QRS_NEXT_CUT()
PTP {E1 29336.919,E2 29336.919}
PTP {X 0,Y 607.923,A -85,B 0,C 180,E1 29336.919,E2 29336.919,E3 0,E4 0,E5 0,E6 0}
QRS_SPEED_INIT()
LIN {X 0,Y 607.923,Z 862.5,A -85,B 0,C 180,E1 29336.919,E2 29336.919,E3 0,E4 0,E5 0,E6 0} C_VEL
LIN {X 0,Y 607.923,Z 712.094,A -85,B 0,C 180,E1 29336.919,E2 29336.919} C_VEL
LIN {X 0,Y 607.923,Z 704.209,A -85,B 0,C 180,E1 29336.919,E2 29336.919} C_VEL
LIN {X 0,Y 607.917,Z 702.213,A -85,B 0,C 180,E1 29336.718,E2 29336.718} C_VEL
LIN {X 0,Y 607.918,Z 702.326,A -85,B 0,C 180,E1 29335.353,E2 29335.353} C_VEL
LIN {X 0,Y 607.916,Z 700.521,A -85,B 0,C 180,E1 29333.863,E2 29333.863} C_VEL
LIN {X 0,Y 607.918,Z 696.809,A -85,B 0,C 180,E1 29332.439,E2 29332.439} C_VEL
LIN {X 0,Y 607.918,Z 691.472,A -85,B 0,C 180,E1 29331.106,E2 29331.106} C_VEL
LIN {X 0,Y 607.918,Z 684.642,A -85,B 0,C 180,E1 29329.864,E2 29329.864} C_VEL
LIN {X 0,Y 607.918,Z 676.351,A -85,B 0,C 180,E1 29328.713,E2 29328.713} C_VEL
LIN {X 0,Y 607.918,Z 666.686,A -85,B 0,C 180,E1 29327.654,E2 29327.654} C_VEL
LIN {X 0,Y 607.92,Z 654.876,A -85,B 0,C 180,E1 29326.639,E2 29326.639} C_VEL
LIN {X 0,Y 607.896,Z 641.663,A -85,B 0,C 180,E1 29325.765,E2 29325.765} C_VEL
LIN {X 0,Y 607.908,Z 627.971,A -85,B 0,C 180,E1 29325.084,E2 29325.084} C_VEL
LIN {X 0,Y 607.9,Z 613.71,A -85,B 0,C 180,E1 29324.571,E2 29324.571} C_VEL
LIN {X 0,Y 607.917,Z 598.614,A -85,B 0,C 180,E1 29324.222,E2 29324.222} C_VEL
LIN {X 0,Y 607.905,Z 485.578,A -85,B 0,C 180,E1 29322.865,E2 29322.865} C_VEL
LIN {X 0,Y 607.912,Z 437.987,A -85,B 0,C 180,E1 29319.693,E2 29319.693} C_VEL
LIN {X 0,Y 607.914,Z 390.758,A -85,B 0,C 180,E1 29316.493,E2 29316.493} C_VEL
LIN {X 0,Y 607.914,Z 343.309,A -85,B 0,C 180,E1 29313.214,E2 29313.214} C_VEL
LIN {X 0,Y 607.918,Z 297.198,A -85,B 0,C 180,E1 29309.949,E2 29309.949} C_VEL
LIN {X 0,Y 607.91,Z 256.209,A -85,B 0,C 180,E1 29307.015,E2 29307.015} C_VEL
LIN {X 0,Y 607.917,Z 237.015,A -85,B 0,C 180,E1 29305.685,E2 29305.685} C_VEL
LIN {X 0,Y 607.9,Z 237.013,A -85,B 0,C 180,E1 29302.514,E2 29302.514} C_VEL
LIN {X 0,Y 607.885,Z 237.014,A -85,B 0,C 180,E1 29299.167,E2 29299.167} C_VEL
LIN {X 0,Y 607.887,Z 237.015,A -85,B 0,C 180,E1 29296.09,E2 29296.09} C_VEL
LIN {X 0,Y 607.912,Z 237.016,A -85,B 0,C 180,E1 29292.916,E2 29292.916} C_VEL
LIN {X 0,Y 607.913,Z 237.011,A -85,B 0,C 180,E1 29289.655,E2 29289.655} C_VEL
LIN {X 0,Y 607.874,Z 237.015,A -85,B 0,C 180,E1 29286.454,E2 29286.454} C_VEL
LIN {X 0,Y 607.914,Z 237.101,A -85,B 0,C 180,E1 29285.87,E2 29285.87} C_VEL
LIN {X 0,Y 607.914,Z 274.11,A -85,B 0,C 180,E1 29282.76,E2 29282.76} C_VEL
LIN {X 0,Y 607.865,Z 300.482,A -85,B 0,C 180,E1 29280.62,E2 29280.62} C_VEL
LIN {X 0,Y 607.913,Z 528.733,A -85,B 0,C 180,E1 29277.674,E2 29277.674} C_VEL
LIN {X 0,Y 607.92,Z 562.49,A -85,B 0,C 180,E1 29277.209,E2 29277.209} C_VEL
LIN {X 0,Y 607.907,Z 582.621,A -85,B 0,C 180,E1 29276.76,E2 29276.76} C_VEL
LIN {X 0,Y 607.907,Z 601.981,A -85,B 0,C 180,E1 29276.155,E2 29276.155} C_VEL
LIN {X 0,Y 607.915,Z 621.48,A -85,B 0,C 180,E1 29275.37,E2 29275.37} C_VEL
LIN {X 0,Y 607.919,Z 640.204,A -85,B 0,C 180,E1 29274.434,E2 29274.434} C_VEL
LIN {X 0,Y 607.916,Z 658.169,A -85,B 0,C 180,E1 29273.352,E2 29273.352} C_VEL
LIN {X 0,Y 607.914,Z 675.868,A -85,B 0,C 180,E1 29272.075,E2 29272.075} C_VEL
LIN {X 0,Y 607.917,Z 692.721,A -85,B 0,C 180,E1 29270.633,E2 29270.633} C_VEL
LIN {X 0,Y 607.908,Z 707.84,A -85,B 0,C 180,E1 29269.106,E2 29269.106} C_VEL
LIN {X 0,Y 607.911,Z 721.188,A -85,B 0,C 180,E1 29267.517,E2 29267.517} C_VEL
LIN {X 0,Y 607.915,Z 733.113,A -85,B 0,C 180,E1 29265.845,E2 29265.845} C_VEL
LIN {X 0,Y 607.91,Z 743.612,A -85,B 0,C 180,E1 29264.089,E2 29264.089} C_VEL
LIN {X 0,Y 607.917,Z 752.375,A -85,B 0,C 180,E1 29262.318,E2 29262.318} C_VEL
LIN {X 0,Y 607.914,Z 759.869,A -85,B 0,C 180,E1 29260.424,E2 29260.424} C_VEL
LIN {X 0,Y 607.913,Z 765.53,A -85,B 0,C 180,E1 29258.513,E2 29258.513} C_VEL
LIN {X 0,Y 607.911,Z 769.46,A -85,B 0,C 180,E1 29256.611,E2 29256.611} C_VEL
LIN {X 0,Y 607.908,Z 771.826,A -85,B 0,C 180,E1 29254.623,E2 29254.623} C_VEL
LIN {X 0,Y 607.906,Z 772.455,A -85,B 0,C 180,E1 29252.734,E2 29252.734} C_VEL
LIN {X 0,Y 607.907,Z 771.512,A -85,B 0,C 180,E1 29250.848,E2 29250.848} C_VEL
LIN {X 0,Y 607.91,Z 768.741,A -85,B 0,C 180,E1 29248.869,E2 29248.869} C_VEL
LIN {X 0,Y 607.912,Z 764.424,A -85,B 0,C 180,E1 29246.983,E2 29246.983} C_VEL
LIN {X 0,Y 607.911,Z 758.417,A -85,B 0,C 180,E1 29245.094,E2 29245.094} C_VEL
LIN {X 0,Y 607.906,Z 751.044,A -85,B 0,C 180,E1 29243.294,E2 29243.294} C_VEL
LIN {X 0,Y 607.906,Z 741.815,A -85,B 0,C 180,E1 29241.487,E2 29241.487} C_VEL
LIN {X 0,Y 607.917,Z 731.146,A -85,B 0,C 180,E1 29239.768,E2 29239.768} C_VEL
LIN {X 0,Y 607.909,Z 719.138,A -85,B 0,C 180,E1 29238.135,E2 29238.135} C_VEL
LIN {X 0,Y 607.913,Z 704.904,A -85,B 0,C 180,E1 29236.494,E2 29236.494} C_VEL
LIN {X 0,Y 607.912,Z 688.936,A -85,B 0,C 180,E1 29234.938,E2 29234.938} C_VEL
LIN {X 0,Y 607.917,Z 672.324,A -85,B 0,C 180,E1 29233.567,E2 29233.567} C_VEL
LIN {X 0,Y 607.919,Z 654.646,A -85,B 0,C 180,E1 29232.335,E2 29232.335} C_VEL
LIN {X 0,Y 607.92,Z 636.895,A -85,B 0,C 180,E1 29231.293,E2 29231.293} C_VEL
LIN {X 0,Y 607.916,Z 617.178,A -85,B 0,C 180,E1 29230.345,E2 29230.345} C_VEL
LIN {X 0,Y 607.918,Z 598.54,A -85,B 0,C 180,E1 29229.636,E2 29229.636} C_VEL
LIN {X 0,Y 607.905,Z 579.176,A -85,B 0,C 180,E1 29229.064,E2 29229.064} C_VEL
LIN {X 0,Y 607.919,Z 559.341,A -85,B 0,C 180,E1 29228.648,E2 29228.648} C_VEL
LIN {X 0,Y 607.901,Z 304.548,A -85,B 0,C 180,E1 29225.345,E2 29225.345} C_VEL
LIN {X 0,Y 607.905,Z 299.084,A -85,B 0,C 180,E1 29225.262,E2 29225.262} C_VEL
LIN {X 0,Y 607.898,Z 255.446,A -85,B 0,C 180,E1 29222.196,E2 29222.196} C_VEL
LIN {X 0,Y 607.906,Z 237.013,A -85,B 0,C 180,E1 29220.853,E2 29220.853} C_VEL
LIN {X 0,Y 607.908,Z 237.015,A -85,B 0,C 180,E1 29217.575,E2 29217.575} C_VEL
LIN {X 0,Y 607.919,Z 237.015,A -85,B 0,C 180,E1 29214.16,E2 29214.16} C_VEL
LIN {X 0,Y 607.891,Z 237.015,A -85,B 0,C 180,E1 29210.953,E2 29210.953} C_VEL
LIN {X 0,Y 607.894,Z 237.015,A -85,B 0,C 180,E1 29207.85,E2 29207.85} C_VEL
LIN {X 0,Y 607.908,Z 237.015,A -85,B 0,C 180,E1 29204.721,E2 29204.721} C_VEL
LIN {X 0,Y 607.889,Z 237.015,A -85,B 0,C 180,E1 29201.519,E2 29201.519} C_VEL
LIN {X 0,Y 607.914,Z 237.013,A -85,B 0,C 180,E1 29198.442,E2 29198.442} C_VEL
LIN {X 0,Y 607.915,Z 237.015,A -85,B 0,C 180,E1 29195.146,E2 29195.146} C_VEL
LIN {X 0,Y 607.915,Z 237.012,A -85,B 0,C 180,E1 29191.868,E2 29191.868} C_VEL
LIN {X 0,Y 607.89,Z 237.015,A -85,B 0,C 180,E1 29188.704,E2 29188.704} C_VEL
LIN {X 0,Y 607.917,Z 237.094,A -85,B 0,C 180,E1 29185.735,E2 29185.735} C_VEL
LIN {X 0,Y 607.912,Z 269.505,A -85,B 0,C 180,E1 29183.25,E2 29183.25} C_VEL
LIN {X 0,Y 607.913,Z 310.074,A -85,B 0,C 180,E1 29180.106,E2 29180.106} C_VEL
LIN {X 0,Y 607.898,Z 351.534,A -85,B 0,C 180,E1 29176.975,E2 29176.975} C_VEL
LIN {X 0,Y 607.914,Z 393.877,A -85,B 0,C 180,E1 29173.846,E2 29173.846} C_VEL
LIN {X 0,Y 607.898,Z 436.137,A -85,B 0,C 180,E1 29170.788,E2 29170.788} C_VEL
LIN {X 0,Y 607.907,Z 578.351,A -85,B 0,C 180,E1 29169.061,E2 29169.061} C_VEL
LIN {X 0,Y 607.914,Z 594.993,A -85,B 0,C 180,E1 29168.677,E2 29168.677} C_VEL
LIN {X 0,Y 607.907,Z 610.686,A -85,B 0,C 180,E1 29168.132,E2 29168.132} C_VEL
LIN {X 0,Y 607.91,Z 625.671,A -85,B 0,C 180,E1 29167.419,E2 29167.419} C_VEL
LIN {X 0,Y 607.919,Z 639.478,A -85,B 0,C 180,E1 29166.576,E2 29166.576} C_VEL
LIN {X 0,Y 607.919,Z 652.518,A -85,B 0,C 180,E1 29165.569,E2 29165.569} C_VEL
LIN {X 0,Y 607.917,Z 664.366,A -85,B 0,C 180,E1 29164.434,E2 29164.434} C_VEL
LIN {X 0,Y 607.919,Z 674.596,A -85,B 0,C 180,E1 29163.206,E2 29163.206} C_VEL
LIN {X 0,Y 607.917,Z 683.39,A -85,B 0,C 180,E1 29161.885,E2 29161.885} C_VEL
LIN {X 0,Y 607.918,Z 690.67,A -85,B 0,C 180,E1 29160.472,E2 29160.472} C_VEL
LIN {X 0,Y 607.914,Z 696.343,A -85,B 0,C 180,E1 29158.964,E2 29158.964} C_VEL
LIN {X 0,Y 607.917,Z 700.143,A -85,B 0,C 180,E1 29157.455,E2 29157.455} C_VEL
LIN {X 0,Y 607.917,Z 702.102,A -85,B 0,C 180,E1 29155.945,E2 29155.945} C_VEL
LIN {X 0,Y 607.916,Z 702.384,A -85,B 0,C 180,E1 29154.432,E2 29154.432} C_VEL
LIN {X 0,Y 607.918,Z 700.91,A -85,B 0,C 180,E1 29152.915,E2 29152.915} C_VEL
LIN {X 0,Y 607.914,Z 697.651,A -85,B 0,C 180,E1 29151.392,E2 29151.392} C_VEL
LIN {X 0,Y 607.914,Z 692.883,A -85,B 0,C 180,E1 29149.96,E2 29149.96} C_VEL
LIN {X 0,Y 607.914,Z 686.165,A -85,B 0,C 180,E1 29148.521,E2 29148.521} C_VEL
LIN {X 0,Y 607.917,Z 677.957,A -85,B 0,C 180,E1 29147.172,E2 29147.172} C_VEL
LIN {X 0,Y 607.917,Z 668.253,A -85,B 0,C 180,E1 29145.912,E2 29145.912} C_VEL
LIN {X 0,Y 607.919,Z 656.49,A -85,B 0,C 180,E1 29144.694,E2 29144.694} C_VEL
LIN {X 0,Y 607.92,Z 644.082,A -85,B 0,C 180,E1 29143.666,E2 29143.666} C_VEL
LIN {X 0,Y 607.904,Z 629.927,A -85,B 0,C 180,E1 29142.73,E2 29142.73} C_VEL
LIN {X 0,Y 607.91,Z 615.562,A -85,B 0,C 180,E1 29141.989,E2 29141.989} C_VEL
LIN {X 0,Y 607.918,Z 600.152,A -85,B 0,C 180,E1 29141.393,E2 29141.393} C_VEL
LIN {X 0,Y 607.911,Z 584.62,A -85,B 0,C 180,E1 29140.97,E2 29140.97} C_VEL
LIN {X 0,Y 607.912,Z 567.42,A -85,B 0,C 180,E1 29140.696,E2 29140.696} C_VEL
LIN {X 0,Y 607.917,Z 435.757,A -85,B 0,C 180,E1 29139.101,E2 29139.101} C_VEL
LIN {X 0,Y 607.898,Z 392.014,A -85,B 0,C 180,E1 29135.927,E2 29135.927} C_VEL
LIN {X 0,Y 607.913,Z 348.895,A -85,B 0,C 180,E1 29132.738,E2 29132.738} C_VEL
LIN {X 0,Y 607.919,Z 306.939,A -85,B 0,C 180,E1 29129.564,E2 29129.564} C_VEL
LIN {X 0,Y 607.907,Z 266.15,A -85,B 0,C 180,E1 29126.396,E2 29126.396} C_VEL
LIN {X 0,Y 607.917,Z 246.516,A -85,B 0,C 180,E1 29124.912,E2 29124.912} C_VEL
LIN {X 0,Y 607.902,Z 237.015,A -85,B 0,C 180,E1 29124.252,E2 29124.252} C_VEL
LIN {X 0,Y 607.914,Z 237.013,A -85,B 0,C 180,E1 29121.075,E2 29121.075} C_VEL
LIN {X 0,Y 607.916,Z 237.209,A -85,B 0,C 180,E1 29119.151,E2 29119.151} C_VEL
LIN {X 0,Y 607.915,Z 286.021,A -85,B 0,C 180,E1 29116.132,E2 29116.132} C_VEL
LIN {X 0,Y 607.892,Z 298.558,A -85,B 0,C 180,E1 29115.28,E2 29115.28} C_VEL
LIN {X 0,Y 607.917,Z 306.589,A -85,B 0,C 180,E1 29114.534,E2 29114.534} C_VEL
LIN {X 0,Y 607.877,Z 311.103,A -85,B 0,C 180,E1 29113.91,E2 29113.91} C_VEL
LIN {X 0,Y 607.877,Z 312.629,A -85,B 0,C 180,E1 29113.436,E2 29113.436} C_VEL
LIN {X 0,Y 607.904,Z 312.223,A -85,B 0,C 180,E1 29113.091,E2 29113.091} C_VEL
LIN {X 0,Y 607.918,Z 310.278,A -85,B 0,C 180,E1 29112.787,E2 29112.787} C_VEL
LIN {X 0,Y 607.903,Z 306.612,A -85,B 0,C 180,E1 29112.532,E2 29112.532} C_VEL
LIN {X 0,Y 607.892,Z 300.365,A -85,B 0,C 180,E1 29112.337,E2 29112.337} C_VEL
LIN {X 0,Y 607.889,Z 290.203,A -85,B 0,C 180,E1 29112.246,E2 29112.246} C_VEL
LIN {X 0,Y 607.888,Z 237.014,A -85,B 0,C 180,E1 29112.229,E2 29112.229} C_VEL
LIN {X 0,Y 607.874,Z 237.015,A -85,B 0,C 180,E1 29109.221,E2 29109.221} C_VEL
LIN {X 0,Y 607.904,Z 237.171,A -85,B 0,C 180,E1 29106.191,E2 29106.191} C_VEL
LIN {X 0,Y 607.917,Z 288.408,A -85,B 0,C 180,E1 29103.158,E2 29103.158} C_VEL
LIN {X 0,Y 607.913,Z 302.276,A -85,B 0,C 180,E1 29102.369,E2 29102.369} C_VEL
LIN {X 0,Y 607.904,Z 524.18,A -85,B 0,C 180,E1 29099.377,E2 29099.377} C_VEL
LIN {X 0,Y 607.903,Z 608.537,A -85,B 0,C 180,E1 29098.234,E2 29098.234} C_VEL
LIN {X 0,Y 607.909,Z 629.043,A -85,B 0,C 180,E1 29097.785,E2 29097.785} C_VEL
LIN {X 0,Y 607.906,Z 649.64,A -85,B 0,C 180,E1 29097.18,E2 29097.18} C_VEL
LIN {X 0,Y 607.913,Z 669.578,A -85,B 0,C 180,E1 29096.417,E2 29096.417} C_VEL
LIN {X 0,Y 607.918,Z 690.744,A -85,B 0,C 180,E1 29095.422,E2 29095.422} C_VEL
LIN {X 0,Y 607.916,Z 710.11,A -85,B 0,C 180,E1 29094.331,E2 29094.331} C_VEL
LIN {X 0,Y 607.914,Z 728.559,A -85,B 0,C 180,E1 29093.096,E2 29093.096} C_VEL
LIN {X 0,Y 607.911,Z 746.777,A -85,B 0,C 180,E1 29091.678,E2 29091.678} C_VEL
LIN {X 0,Y 607.913,Z 763.653,A -85,B 0,C 180,E1 29090.156,E2 29090.156} C_VEL
LIN {X 0,Y 607.918,Z 779.465,A -85,B 0,C 180,E1 29088.508,E2 29088.508} C_VEL
LIN {X 0,Y 607.913,Z 793.413,A -85,B 0,C 180,E1 29086.817,E2 29086.817} C_VEL
LIN {X 0,Y 607.918,Z 805.901,A -85,B 0,C 180,E1 29085.062,E2 29085.062} C_VEL
LIN {X 0,Y 607.919,Z 817.421,A -85,B 0,C 180,E1 29083.176,E2 29083.176} C_VEL
LIN {X 0,Y 607.912,Z 827.061,A -85,B 0,C 180,E1 29081.287,E2 29081.287} C_VEL
LIN {X 0,Y 607.911,Z 835.464,A -85,B 0,C 180,E1 29079.276,E2 29079.276} C_VEL
LIN {X 0,Y 607.91,Z 842.129,A -85,B 0,C 180,E1 29077.276,E2 29077.276} C_VEL
LIN {X 0,Y 607.912,Z 847.015,A -85,B 0,C 180,E1 29075.285,E2 29075.285} C_VEL
LIN {X 0,Y 607.917,Z 850.447,A -85,B 0,C 180,E1 29073.206,E2 29073.206} C_VEL
LIN {X 0,Y 607.91,Z 852.21,A -85,B 0,C 180,E1 29071.225,E2 29071.225} C_VEL
LIN {X 0,Y 607.902,Z 852.329,A -85,B 0,C 180,E1 29069.246,E2 29069.246} C_VEL
LIN {X 0,Y 607.908,Z 850.896,A -85,B 0,C 180,E1 29067.172,E2 29067.172} C_VEL
LIN {X 0,Y 607.912,Z 847.987,A -85,B 0,C 180,E1 29065.188,E2 29065.188} C_VEL
LIN {X 0,Y 607.915,Z 843.399,A -85,B 0,C 180,E1 29063.199,E2 29063.199} C_VEL
LIN {X 0,Y 607.906,Z 837.238,A -85,B 0,C 180,E1 29061.201,E2 29061.201} C_VEL
LIN {X 0,Y 607.899,Z 829.657,A -85,B 0,C 180,E1 29059.289,E2 29059.289} C_VEL
LIN {X 0,Y 607.899,Z 820.326,A -85,B 0,C 180,E1 29057.364,E2 29057.364} C_VEL
LIN {X 0,Y 607.904,Z 809.744,A -85,B 0,C 180,E1 29055.522,E2 29055.522} C_VEL
LIN {X 0,Y 607.913,Z 797.033,A -85,B 0,C 180,E1 29053.665,E2 29053.665} C_VEL
LIN {X 0,Y 607.907,Z 782.865,A -85,B 0,C 180,E1 29051.889,E2 29051.889} C_VEL
LIN {X 0,Y 607.91,Z 767.096,A -85,B 0,C 180,E1 29050.185,E2 29050.185} C_VEL
LIN {X 0,Y 607.918,Z 750.497,A -85,B 0,C 180,E1 29048.635,E2 29048.635} C_VEL
LIN {X 0,Y 607.913,Z 732.133,A -85,B 0,C 180,E1 29047.16,E2 29047.16} C_VEL
LIN {X 0,Y 607.915,Z 713.681,A -85,B 0,C 180,E1 29045.898,E2 29045.898} C_VEL
LIN {X 0,Y 607.918,Z 693.554,A -85,B 0,C 180,E1 29044.726,E2 29044.726} C_VEL
LIN {X 0,Y 607.904,Z 674.553,A -85,B 0,C 180,E1 29043.792,E2 29043.792} C_VEL
LIN {X 0,Y 607.906,Z 653.962,A -85,B 0,C 180,E1 29042.976,E2 29042.976} C_VEL
LIN {X 0,Y 607.917,Z 632.86,A -85,B 0,C 180,E1 29042.313,E2 29042.313} C_VEL
LIN {X 0,Y 607.905,Z 613.424,A -85,B 0,C 180,E1 29041.861,E2 29041.861} C_VEL
LIN {X 0,Y 607.918,Z 585.551,A -85,B 0,C 180,E1 29041.436,E2 29041.436} C_VEL
LIN {X 0,Y 607.876,Z 362.254,A -85,B 0,C 180,E1 29038.447,E2 29038.447} C_VEL
LIN {X 0,Y 607.915,Z 302.732,A -85,B 0,C 180,E1 29037.631,E2 29037.631} C_VEL
LIN {X 0,Y 607.898,Z 258.862,A -85,B 0,C 180,E1 29034.622,E2 29034.622} C_VEL
LIN {X 0,Y 607.893,Z 237.014,A -85,B 0,C 180,E1 29033.07,E2 29033.07} C_VEL
LIN {X 0,Y 607.882,Z 237.015,A -85,B 0,C 180,E1 29029.974,E2 29029.974} C_VEL
LIN {X 0,Y 607.902,Z 237.013,A -85,B 0,C 180,E1 29027.753,E2 29027.753} C_VEL
LIN {X 0,Y 607.902,Z 333.704,A -85,B 0,C 180,E1 29027.733,E2 29027.733} C_VEL
LIN {X 0,Y 607.904,Z 341.134,A -85,B 0,C 180,E1 29027.596,E2 29027.596} C_VEL
LIN {X 0,Y 607.909,Z 345.398,A -85,B 0,C 180,E1 29027.402,E2 29027.402} C_VEL
LIN {X 0,Y 607.917,Z 347.912,A -85,B 0,C 180,E1 29027.184,E2 29027.184} C_VEL
LIN {X 0,Y 607.917,Z 349.732,A -85,B 0,C 180,E1 29026.826,E2 29026.826} C_VEL
LIN {X 0,Y 607.884,Z 349.905,A -85,B 0,C 180,E1 29026.434,E2 29026.434} C_VEL
LIN {X 0,Y 607.884,Z 348.098,A -85,B 0,C 180,E1 29025.912,E2 29025.912} C_VEL
LIN {X 0,Y 607.915,Z 343.085,A -85,B 0,C 180,E1 29025.199,E2 29025.199} C_VEL
LIN {X 0,Y 607.899,Z 335.413,A -85,B 0,C 180,E1 29024.452,E2 29024.452} C_VEL
LIN {X 0,Y 607.906,Z 321.424,A -85,B 0,C 180,E1 29023.433,E2 29023.433} C_VEL
LIN {X 0,Y 607.911,Z 279.23,A -85,B 0,C 180,E1 29020.459,E2 29020.459} C_VEL
LIN {X 0,Y 607.895,Z 240.537,A -85,B 0,C 180,E1 29017.605,E2 29017.605} C_VEL
LIN {X 0,Y 607.917,Z 237.015,A -85,B 0,C 180,E1 29017.336,E2 29017.336} C_VEL
LIN {X 0,Y 607.89,Z 237.014,A -85,B 0,C 180,E1 29014.173,E2 29014.173} C_VEL
LIN {X 0,Y 607.911,Z 237.007,A -85,B 0,C 180,E1 29010.874,E2 29010.874} C_VEL
LIN {X 0,Y 607.873,Z 237.012,A -85,B 0,C 180,E1 29007.742,E2 29007.742} C_VEL
LIN {X 0,Y 607.866,Z 237.166,A -85,B 0,C 180,E1 29006.08,E2 29006.08} C_VEL
LIN {X 0,Y 607.91,Z 268.682,A -85,B 0,C 180,E1 29004.021,E2 29004.021} C_VEL
LIN {X 0,Y 607.911,Z 313.328,A -85,B 0,C 180,E1 29000.809,E2 29000.809} C_VEL
LIN {X 0,Y 607.913,Z 359.543,A -85,B 0,C 180,E1 28997.566,E2 28997.566} C_VEL
LIN {X 0,Y 607.912,Z 407.398,A -85,B 0,C 180,E1 28994.283,E2 28994.283} C_VEL
LIN {X 0,Y 607.915,Z 454.742,A -85,B 0,C 180,E1 28991.095,E2 28991.095} C_VEL
LIN {X 0,Y 607.91,Z 485.669,A -85,B 0,C 180,E1 28989.043,E2 28989.043} C_VEL
LIN {X 0,Y 607.919,Z 599.073,A -85,B 0,C 180,E1 28987.679,E2 28987.679} C_VEL
LIN {X 0,Y 607.903,Z 613.667,A -85,B 0,C 180,E1 28987.34,E2 28987.34} C_VEL
LIN {X 0,Y 607.908,Z 627.464,A -85,B 0,C 180,E1 28986.848,E2 28986.848} C_VEL
LIN {X 0,Y 607.897,Z 640.982,A -85,B 0,C 180,E1 28986.184,E2 28986.184} C_VEL
LIN {X 0,Y 607.918,Z 654.051,A -85,B 0,C 180,E1 28985.332,E2 28985.332} C_VEL
LIN {X 0,Y 607.919,Z 665.313,A -85,B 0,C 180,E1 28984.386,E2 28984.386} C_VEL
LIN {X 0,Y 607.917,Z 674.746,A -85,B 0,C 180,E1 28983.394,E2 28983.394} C_VEL
LIN {X 0,Y 607.918,Z 683.863,A -85,B 0,C 180,E1 28982.168,E2 28982.168} C_VEL
LIN {X 0,Y 607.918,Z 690.803,A -85,B 0,C 180,E1 28980.942,E2 28980.942} C_VEL
LIN {X 0,Y 607.919,Z 696.321,A -85,B 0,C 180,E1 28979.623,E2 28979.623} C_VEL
LIN {X 0,Y 607.916,Z 700.179,A -85,B 0,C 180,E1 28978.209,E2 28978.209} C_VEL
LIN {X 0,Y 607.916,Z 702.093,A -85,B 0,C 180,E1 28976.888,E2 28976.888} C_VEL
LIN {X 0,Y 607.917,Z 702.213,A -85,B 0,C 180,E1 28976.718,E2 28976.718} C_VEL
LIN {X 0,Y 606.916,Z 702.497,A -85,B 0,C 180,E1 28975.992,E2 28975.992} C_VEL
LIN {X 0,Y 602.995,Z 701.936,A -85,B 0,C 180,E1 28974.831,E2 28974.831} C_VEL
LIN {X 0,Y 600.268,Z 700.564,A -85,B 0,C 180,E1 28973.859,E2 28973.859} C_VEL
LIN {X 0,Y 599.917,Z 699.685,A -85,B 0,C 180,E1 28973.441,E2 28973.441} C_VEL
LIN {X 0,Y 599.916,Z 695.635,A -85,B 0,C 180,E1 28972.048,E2 28972.048} C_VEL
LIN {X 0,Y 599.922,Z 689.797,A -85,B 0,C 180,E1 28970.696,E2 28970.696} C_VEL
LIN {X 0,Y 599.932,Z 682.383,A -85,B 0,C 180,E1 28969.436,E2 28969.436} C_VEL
LIN {X 0,Y 599.948,Z 673.454,A -85,B 0,C 180,E1 28968.268,E2 28968.268} C_VEL
LIN {X 0,Y 599.971,Z 663.013,A -85,B 0,C 180,E1 28967.194,E2 28967.194} C_VEL
LIN {X 0,Y 599.986,Z 650.76,A -85,B 0,C 180,E1 28966.213,E2 28966.213} C_VEL
LIN {X 0,Y 600.002,Z 638.006,A -85,B 0,C 180,E1 28965.426,E2 28965.426} C_VEL
LIN {X 0,Y 600.029,Z 624.106,A -85,B 0,C 180,E1 28964.779,E2 28964.779} C_VEL
LIN {X 0,Y 600.056,Z 609.272,A -85,B 0,C 180,E1 28964.296,E2 28964.296} C_VEL
LIN {X 0,Y 600.085,Z 594.128,A -85,B 0,C 180,E1 28963.999,E2 28963.999} C_VEL
LIN {X 0,Y 600.045,Z 485.282,A -85,B 0,C 180,E1 28962.671,E2 28962.671} C_VEL
LIN {X 0,Y 600.129,Z 438.627,A -85,B 0,C 180,E1 28959.52,E2 28959.52} C_VEL
LIN {X 0,Y 600.229,Z 391.488,A -85,B 0,C 180,E1 28956.285,E2 28956.285} C_VEL
LIN {X 0,Y 600.333,Z 343.943,A -85,B 0,C 180,E1 28952.955,E2 28952.955} C_VEL
LIN {X 0,Y 600.463,Z 298.529,A -85,B 0,C 180,E1 28949.699,E2 28949.699} C_VEL
LIN {X 0,Y 600.322,Z 250.637,A -85,B 0,C 180,E1 28946.315,E2 28946.315} C_VEL
LIN {X 0,Y 600.245,Z 239.331,A -85,B 0,C 180,E1 28945.543,E2 28945.543} C_VEL
LIN {X 0,Y 599.953,Z 238.005,A -85,B 0,C 180,E1 28945.415,E2 28945.415} C_VEL
LIN {X 0,Y 599.96,Z 238,A -85,B 0,C 180,E1 28942.293,E2 28942.293} C_VEL
LIN {X 0,Y 599.952,Z 238.003,A -85,B 0,C 180,E1 28938.956,E2 28938.956} C_VEL
LIN {X 0,Y 599.976,Z 238.004,A -85,B 0,C 180,E1 28935.775,E2 28935.775} C_VEL
LIN {X 0,Y 599.951,Z 238.004,A -85,B 0,C 180,E1 28932.555,E2 28932.555} C_VEL
LIN {X 0,Y 599.959,Z 238.002,A -85,B 0,C 180,E1 28929.17,E2 28929.17} C_VEL
LIN {X 0,Y 599.959,Z 238.135,A -85,B 0,C 180,E1 28926.273,E2 28926.273} C_VEL
LIN {X 0,Y 600.701,Z 241.601,A -85,B 0,C 180,E1 28925.926,E2 28925.926} C_VEL
LIN {X 0,Y 600.543,Z 278.735,A -85,B 0,C 180,E1 28922.776,E2 28922.776} C_VEL
LIN {X 0,Y 600.532,Z 300.692,A -85,B 0,C 180,E1 28920.985,E2 28920.985} C_VEL
LIN {X 0,Y 600.761,Z 314.388,A -85,B 0,C 180,E1 28920.792,E2 28920.792} C_VEL
LIN {X 0,Y 600.62,Z 561.056,A -85,B 0,C 180,E1 28917.551,E2 28917.551} C_VEL
LIN {X 0,Y 600.559,Z 581.248,A -85,B 0,C 180,E1 28917.104,E2 28917.104} C_VEL
LIN {X 0,Y 600.497,Z 601.492,A -85,B 0,C 180,E1 28916.476,E2 28916.476} C_VEL
LIN {X 0,Y 600.424,Z 621.676,A -85,B 0,C 180,E1 28915.656,E2 28915.656} C_VEL
LIN {X 0,Y 600.344,Z 640.35,A -85,B 0,C 180,E1 28914.711,E2 28914.711} C_VEL
LIN {X 0,Y 600.274,Z 658.008,A -85,B 0,C 180,E1 28913.634,E2 28913.634} C_VEL
LIN {X 0,Y 600.199,Z 675.975,A -85,B 0,C 180,E1 28912.323,E2 28912.323} C_VEL
LIN {X 0,Y 600.123,Z 692.516,A -85,B 0,C 180,E1 28910.888,E2 28910.888} C_VEL
LIN {X 0,Y 600.061,Z 707.447,A -85,B 0,C 180,E1 28909.365,E2 28909.365} C_VEL
LIN {X 0,Y 600.006,Z 720.857,A -85,B 0,C 180,E1 28907.756,E2 28907.756} C_VEL
LIN {X 0,Y 599.976,Z 732.845,A -85,B 0,C 180,E1 28906.06,E2 28906.06} C_VEL
LIN {X 0,Y 599.948,Z 743.391,A -85,B 0,C 180,E1 28904.28,E2 28904.28} C_VEL
LIN {X 0,Y 599.929,Z 752.089,A -85,B 0,C 180,E1 28902.513,E2 28902.513} C_VEL
LIN {X 0,Y 599.923,Z 759.729,A -85,B 0,C 180,E1 28900.564,E2 28900.564} C_VEL
LIN {X 0,Y 599.917,Z 765.422,A -85,B 0,C 180,E1 28898.627,E2 28898.627} C_VEL
LIN {X 0,Y 599.914,Z 769.398,A -85,B 0,C 180,E1 28896.7,E2 28896.7} C_VEL
LIN {X 0,Y 599.91,Z 771.811,A -85,B 0,C 180,E1 28894.668,E2 28894.668} C_VEL
LIN {X 0,Y 599.907,Z 772.466,A -85,B 0,C 180,E1 28892.77,E2 28892.77} C_VEL
LIN {X 0,Y 599.904,Z 771.452,A -85,B 0,C 180,E1 28890.764,E2 28890.764} C_VEL
LIN {X 0,Y 599.91,Z 768.805,A -85,B 0,C 180,E1 28888.854,E2 28888.854} C_VEL
LIN {X 0,Y 599.914,Z 764.532,A -85,B 0,C 180,E1 28886.943,E2 28886.943} C_VEL
LIN {X 0,Y 599.921,Z 758.565,A -85,B 0,C 180,E1 28885.028,E2 28885.028} C_VEL
LIN {X 0,Y 599.925,Z 751.236,A -85,B 0,C 180,E1 28883.204,E2 28883.204} C_VEL
LIN {X 0,Y 599.94,Z 742.034,A -85,B 0,C 180,E1 28881.373,E2 28881.373} C_VEL
LIN {X 0,Y 599.977,Z 731.414,A -85,B 0,C 180,E1 28879.631,E2 28879.631} C_VEL
LIN {X 0,Y 600.011,Z 719.467,A -85,B 0,C 180,E1 28877.977,E2 28877.977} C_VEL
LIN {X 0,Y 600.067,Z 705.293,A -85,B 0,C 180,E1 28876.314,E2 28876.314} C_VEL
LIN {X 0,Y 600.128,Z 689.941,A -85,B 0,C 180,E1 28874.787,E2 28874.787} C_VEL
LIN {X 0,Y 600.205,Z 673.528,A -85,B 0,C 180,E1 28873.399,E2 28873.399} C_VEL
LIN {X 0,Y 600.288,Z 656.096,A -85,B 0,C 180,E1 28872.153,E2 28872.153} C_VEL
LIN {X 0,Y 600.367,Z 637.68,A -85,B 0,C 180,E1 28871.049,E2 28871.049} C_VEL
LIN {X 0,Y 600.439,Z 618.129,A -85,B 0,C 180,E1 28870.09,E2 28870.09} C_VEL
LIN {X 0,Y 600.509,Z 599.057,A -85,B 0,C 180,E1 28869.349,E2 28869.349} C_VEL
LIN {X 0,Y 600.563,Z 578.722,A -85,B 0,C 180,E1 28868.741,E2 28868.741} C_VEL
LIN {X 0,Y 600.621,Z 558.236,A -85,B 0,C 180,E1 28868.316,E2 28868.316} C_VEL
LIN {X 0,Y 600.809,Z 305.225,A -85,B 0,C 180,E1 28864.999,E2 28864.999} C_VEL
LIN {X 0,Y 600.554,Z 299.244,A -85,B 0,C 180,E1 28864.905,E2 28864.905} C_VEL
LIN {X 0,Y 600.676,Z 255.491,A -85,B 0,C 180,E1 28861.788,E2 28861.788} C_VEL
LIN {X 0,Y 600.531,Z 240.103,A -85,B 0,C 180,E1 28860.656,E2 28860.656} C_VEL
LIN {X 0,Y 599.979,Z 238.001,A -85,B 0,C 180,E1 28860.443,E2 28860.443} C_VEL
LIN {X 0,Y 599.953,Z 238.004,A -85,B 0,C 180,E1 28857.312,E2 28857.312} C_VEL
LIN {X 0,Y 599.975,Z 238.005,A -85,B 0,C 180,E1 28854.083,E2 28854.083} C_VEL
LIN {X 0,Y 599.952,Z 238.005,A -85,B 0,C 180,E1 28850.952,E2 28850.952} C_VEL
LIN {X 0,Y 599.953,Z 238.004,A -85,B 0,C 180,E1 28847.807,E2 28847.807} C_VEL
LIN {X 0,Y 599.976,Z 238.004,A -85,B 0,C 180,E1 28844.635,E2 28844.635} C_VEL
LIN {X 0,Y 599.961,Z 238.003,A -85,B 0,C 180,E1 28841.27,E2 28841.27} C_VEL
LIN {X 0,Y 599.978,Z 238,A -85,B 0,C 180,E1 28838.069,E2 28838.069} C_VEL
LIN {X 0,Y 599.965,Z 238.003,A -85,B 0,C 180,E1 28834.864,E2 28834.864} C_VEL
LIN {X 0,Y 599.973,Z 238.004,A -85,B 0,C 180,E1 28831.553,E2 28831.553} C_VEL
LIN {X 0,Y 599.953,Z 238.004,A -85,B 0,C 180,E1 28828.358,E2 28828.358} C_VEL
LIN {X 0,Y 599.981,Z 238.047,A -85,B 0,C 180,E1 28825.995,E2 28825.995} C_VEL
LIN {X 0,Y 600.345,Z 242.342,A -85,B 0,C 180,E1 28825.66,E2 28825.66} C_VEL
LIN {X 0,Y 600.484,Z 284.835,A -85,B 0,C 180,E1 28822.415,E2 28822.415} C_VEL
LIN {X 0,Y 600.35,Z 325.484,A -85,B 0,C 180,E1 28819.255,E2 28819.255} C_VEL
LIN {X 0,Y 600.255,Z 367.017,A -85,B 0,C 180,E1 28816.102,E2 28816.102} C_VEL
LIN {X 0,Y 600.148,Z 409.648,A -85,B 0,C 180,E1 28812.934,E2 28812.934} C_VEL
LIN {X 0,Y 600.155,Z 436.538,A -85,B 0,C 180,E1 28810.993,E2 28810.993} C_VEL
LIN {X 0,Y 600.143,Z 578.774,A -85,B 0,C 180,E1 28809.24,E2 28809.24} C_VEL
LIN {X 0,Y 600.129,Z 595.596,A -85,B 0,C 180,E1 28808.842,E2 28808.842} C_VEL
LIN {X 0,Y 600.088,Z 611.149,A -85,B 0,C 180,E1 28808.287,E2 28808.287} C_VEL
LIN {X 0,Y 600.053,Z 627.239,A -85,B 0,C 180,E1 28807.499,E2 28807.499} C_VEL
LIN {X 0,Y 600.024,Z 641.272,A -85,B 0,C 180,E1 28806.603,E2 28806.603} C_VEL
LIN {X 0,Y 599.992,Z 655.087,A -85,B 0,C 180,E1 28805.485,E2 28805.485} C_VEL
LIN {X 0,Y 599.962,Z 666.654,A -85,B 0,C 180,E1 28804.301,E2 28804.301} C_VEL
LIN {X 0,Y 599.942,Z 676.488,A -85,B 0,C 180,E1 28803.057,E2 28803.057} C_VEL
LIN {X 0,Y 599.927,Z 684.842,A -85,B 0,C 180,E1 28801.719,E2 28801.719} C_VEL
LIN {X 0,Y 599.92,Z 691.759,A -85,B 0,C 180,E1 28800.287,E2 28800.287} C_VEL
LIN {X 0,Y 599.916,Z 697.135,A -85,B 0,C 180,E1 28798.759,E2 28798.759} C_VEL
LIN {X 0,Y 599.915,Z 700.568,A -85,B 0,C 180,E1 28797.23,E2 28797.23} C_VEL
LIN {X 0,Y 599.914,Z 702.345,A -85,B 0,C 180,E1 28795.603,E2 28795.603} C_VEL
LIN {X 0,Y 599.915,Z 702.177,A -85,B 0,C 180,E1 28794.069,E2 28794.069} C_VEL
LIN {X 0,Y 599.915,Z 700.322,A -85,B 0,C 180,E1 28792.531,E2 28792.531} C_VEL
LIN {X 0,Y 599.916,Z 696.636,A -85,B 0,C 180,E1 28790.987,E2 28790.987} C_VEL
LIN {X 0,Y 599.919,Z 691.338,A -85,B 0,C 180,E1 28789.525,E2 28789.525} C_VEL
LIN {X 0,Y 599.929,Z 684.221,A -85,B 0,C 180,E1 28788.074,E2 28788.074} C_VEL
LIN {X 0,Y 599.945,Z 675.393,A -85,B 0,C 180,E1 28786.704,E2 28786.704} C_VEL
LIN {X 0,Y 599.965,Z 665.048,A -85,B 0,C 180,E1 28785.425,E2 28785.425} C_VEL
LIN {X 0,Y 599.995,Z 652.968,A -85,B 0,C 180,E1 28784.239,E2 28784.239} C_VEL
LIN {X 0,Y 600.024,Z 640.4,A -85,B 0,C 180,E1 28783.245,E2 28783.245} C_VEL
LIN {X 0,Y 600.054,Z 626.791,A -85,B 0,C 180,E1 28782.387,E2 28782.387} C_VEL
LIN {X 0,Y 600.086,Z 611.637,A -85,B 0,C 180,E1 28781.645,E2 28781.645} C_VEL
LIN {X 0,Y 600.129,Z 596.071,A -85,B 0,C 180,E1 28781.083,E2 28781.083} C_VEL
LIN {X 0,Y 600.145,Z 579.592,A -85,B 0,C 180,E1 28780.685,E2 28780.685} C_VEL
LIN {X 0,Y 600.176,Z 538.532,A -85,B 0,C 180,E1 28780.158,E2 28780.158} C_VEL
LIN {X 0,Y 600.114,Z 436,A -85,B 0,C 180,E1 28778.907,E2 28778.907} C_VEL
LIN {X 0,Y 600.182,Z 393.117,A -85,B 0,C 180,E1 28775.755,E2 28775.755} C_VEL
LIN {X 0,Y 600.295,Z 350.929,A -85,B 0,C 180,E1 28772.595,E2 28772.595} C_VEL
LIN {X 0,Y 600.415,Z 308.75,A -85,B 0,C 180,E1 28769.365,E2 28769.365} C_VEL
LIN {X 0,Y 600.429,Z 271.807,A -85,B 0,C 180,E1 28766.494,E2 28766.494} C_VEL
LIN {X 0,Y 599.96,Z 238.004,A -85,B 0,C 180,E1 28764.171,E2 28764.171} C_VEL
LIN {X 0,Y 599.978,Z 238.001,A -85,B 0,C 180,E1 28760.95,E2 28760.95} C_VEL
LIN {X 0,Y 599.977,Z 238.162,A -85,B 0,C 180,E1 28759.738,E2 28759.738} C_VEL
LIN {X 0,Y 601.386,Z 241.742,A -85,B 0,C 180,E1 28759.391,E2 28759.391} C_VEL
LIN {X 0,Y 601.191,Z 290.6,A -85,B 0,C 180,E1 28756.341,E2 28756.341} C_VEL
LIN {X 0,Y 601.878,Z 304.835,A -85,B 0,C 180,E1 28755.423,E2 28755.423} C_VEL
LIN {X 0,Y 602.923,Z 312.502,A -85,B 0,C 180,E1 28754.784,E2 28754.784} C_VEL
LIN {X 0,Y 603.87,Z 317.346,A -85,B 0,C 180,E1 28754.193,E2 28754.193} C_VEL
LIN {X 0,Y 604.594,Z 319.521,A -85,B 0,C 180,E1 28753.723,E2 28753.723} C_VEL
LIN {X 0,Y 605.181,Z 320.146,A -85,B 0,C 180,E1 28753.231,E2 28753.231} C_VEL
LIN {X 0,Y 605.41,Z 318.965,A -85,B 0,C 180,E1 28752.749,E2 28752.749} C_VEL
LIN {X 0,Y 605.162,Z 316.09,A -85,B 0,C 180,E1 28752.337,E2 28752.337} C_VEL
LIN {X 0,Y 604.488,Z 311.563,A -85,B 0,C 180,E1 28752.011,E2 28752.011} C_VEL
LIN {X 0,Y 603.535,Z 305.051,A -85,B 0,C 180,E1 28751.795,E2 28751.795} C_VEL
LIN {X 0,Y 602.626,Z 294.653,A -85,B 0,C 180,E1 28751.692,E2 28751.692} C_VEL
LIN {X 0,Y 602.377,Z 242.797,A -85,B 0,C 180,E1 28751.665,E2 28751.665} C_VEL
LIN {X 0,Y 600.469,Z 239.953,A -85,B 0,C 180,E1 28751.46,E2 28751.46} C_VEL
LIN {X 0,Y 599.973,Z 238.003,A -85,B 0,C 180,E1 28751.389,E2 28751.389} C_VEL
LIN {X 0,Y 599.94,Z 238.005,A -85,B 0,C 180,E1 28748.193,E2 28748.193} C_VEL
LIN {X 0,Y 599.98,Z 238.019,A -85,B 0,C 180,E1 28746.694,E2 28746.694} C_VEL
LIN {X 0,Y 601.097,Z 241.818,A -85,B 0,C 180,E1 28746.382,E2 28746.382} C_VEL
LIN {X 0,Y 600.926,Z 292.429,A -85,B 0,C 180,E1 28743.358,E2 28743.358} C_VEL
LIN {X 0,Y 601.014,Z 302.701,A -85,B 0,C 180,E1 28742.781,E2 28742.781} C_VEL
LIN {X 0,Y 600.96,Z 495.848,A -85,B 0,C 180,E1 28740.133,E2 28740.133} C_VEL
LIN {X 0,Y 600.847,Z 608.558,A -85,B 0,C 180,E1 28738.596,E2 28738.596} C_VEL
LIN {X 0,Y 600.79,Z 629.726,A -85,B 0,C 180,E1 28738.126,E2 28738.126} C_VEL
LIN {X 0,Y 600.703,Z 651.089,A -85,B 0,C 180,E1 28737.481,E2 28737.481} C_VEL
LIN {X 0,Y 600.638,Z 671.563,A -85,B 0,C 180,E1 28736.68,E2 28736.68} C_VEL
LIN {X 0,Y 600.538,Z 691.744,A -85,B 0,C 180,E1 28735.704,E2 28735.704} C_VEL
LIN {X 0,Y 600.434,Z 710.925,A -85,B 0,C 180,E1 28734.602,E2 28734.602} C_VEL
LIN {X 0,Y 600.348,Z 730.016,A -85,B 0,C 180,E1 28733.3,E2 28733.3} C_VEL
LIN {X 0,Y 600.246,Z 747.555,A -85,B 0,C 180,E1 28731.903,E2 28731.903} C_VEL
LIN {X 0,Y 600.16,Z 765.176,A -85,B 0,C 180,E1 28730.275,E2 28730.275} C_VEL
LIN {X 0,Y 600.091,Z 780.318,A -85,B 0,C 180,E1 28728.657,E2 28728.657} C_VEL
LIN {X 0,Y 600.038,Z 794.885,A -85,B 0,C 180,E1 28726.855,E2 28726.855} C_VEL
LIN {X 0,Y 599.994,Z 807.187,A -85,B 0,C 180,E1 28725.068,E2 28725.068} C_VEL
LIN {X 0,Y 599.956,Z 818.772,A -85,B 0,C 180,E1 28723.1,E2 28723.1} C_VEL
LIN {X 0,Y 599.94,Z 828.43,A -85,B 0,C 180,E1 28721.147,E2 28721.147} C_VEL
LIN {X 0,Y 599.928,Z 836.176,A -85,B 0,C 180,E1 28719.207,E2 28719.207} C_VEL
LIN {X 0,Y 599.922,Z 842.894,A -85,B 0,C 180,E1 28717.084,E2 28717.084} C_VEL
LIN {X 0,Y 599.917,Z 847.635,A -85,B 0,C 180,E1 28715.068,E2 28715.068} C_VEL
LIN {X 0,Y 599.914,Z 850.786,A -85,B 0,C 180,E1 28712.962,E2 28712.962} C_VEL
LIN {X 0,Y 599.903,Z 852.332,A -85,B 0,C 180,E1 28710.764,E2 28710.764} C_VEL
LIN {X 0,Y 599.907,Z 852.209,A -85,B 0,C 180,E1 28708.758,E2 28708.758} C_VEL
LIN {X 0,Y 599.916,Z 850.373,A -85,B 0,C 180,E1 28706.686,E2 28706.686} C_VEL
LIN {X 0,Y 599.915,Z 846.812,A -85,B 0,C 180,E1 28704.549,E2 28704.549} C_VEL
LIN {X 0,Y 599.912,Z 841.871,A -85,B 0,C 180,E1 28702.53,E2 28702.53} C_VEL
LIN {X 0,Y 599.915,Z 835.112,A -85,B 0,C 180,E1 28700.503,E2 28700.503} C_VEL
LIN {X 0,Y 599.93,Z 826.601,A -85,B 0,C 180,E1 28698.463,E2 28698.463} C_VEL
LIN {X 0,Y 599.958,Z 816.689,A -85,B 0,C 180,E1 28696.507,E2 28696.507} C_VEL
LIN {X 0,Y 599.998,Z 805.263,A -85,B 0,C 180,E1 28694.635,E2 28694.635} C_VEL
LIN {X 0,Y 600.05,Z 791.786,A -85,B 0,C 180,E1 28692.746,E2 28692.746} C_VEL
LIN {X 0,Y 600.103,Z 777.668,A -85,B 0,C 180,E1 28691.04,E2 28691.04} C_VEL
LIN {X 0,Y 600.181,Z 761.624,A -85,B 0,C 180,E1 28689.369,E2 28689.369} C_VEL
LIN {X 0,Y 600.259,Z 744.53,A -85,B 0,C 180,E1 28687.84,E2 28687.84} C_VEL
LIN {X 0,Y 600.363,Z 726.38,A -85,B 0,C 180,E1 28686.44,E2 28686.44} C_VEL
LIN {X 0,Y 600.469,Z 707.039,A -85,B 0,C 180,E1 28685.161,E2 28685.161} C_VEL
LIN {X 0,Y 600.551,Z 687.767,A -85,B 0,C 180,E1 28684.085,E2 28684.085} C_VEL
LIN {X 0,Y 600.653,Z 667.609,A -85,B 0,C 180,E1 28683.155,E2 28683.155} C_VEL
LIN {X 0,Y 600.74,Z 646.81,A -85,B 0,C 180,E1 28682.374,E2 28682.374} C_VEL
LIN {X 0,Y 600.794,Z 625.997,A -85,B 0,C 180,E1 28681.777,E2 28681.777} C_VEL
LIN {X 0,Y 600.858,Z 604.27,A -85,B 0,C 180,E1 28681.336,E2 28681.336} C_VEL
LIN {X 0,Y 601.051,Z 369.197,A -85,B 0,C 180,E1 28678.143,E2 28678.143} C_VEL
LIN {X 0,Y 600.957,Z 303.555,A -85,B 0,C 180,E1 28677.228,E2 28677.228} C_VEL
LIN {X 0,Y 600.818,Z 299.504,A -85,B 0,C 180,E1 28676.98,E2 28676.98} C_VEL
LIN {X 0,Y 600.957,Z 257.206,A -85,B 0,C 180,E1 28674.033,E2 28674.033} C_VEL
LIN {X 0,Y 600.856,Z 240.834,A -85,B 0,C 180,E1 28672.852,E2 28672.852} C_VEL
LIN {X 0,Y 599.951,Z 238.005,A -85,B 0,C 180,E1 28672.578,E2 28672.578} C_VEL
LIN {X 0,Y 599.977,Z 238.004,A -85,B 0,C 180,E1 28669.457,E2 28669.457} C_VEL
LIN {X 0,Y 599.965,Z 238.098,A -85,B 0,C 180,E1 28668.594,E2 28668.594} C_VEL
LIN {X 0,Y 601.05,Z 241.154,A -85,B 0,C 180,E1 28668.477,E2 28668.477} C_VEL
LIN {X 0,Y 602.551,Z 242.959,A -85,B 0,C 180,E1 28668.316,E2 28668.316} C_VEL
LIN {X 0,Y 602.731,Z 335.454,A -85,B 0,C 180,E1 28668.297,E2 28668.297} C_VEL
LIN {X 0,Y 603.698,Z 344.274,A -85,B 0,C 180,E1 28668.173,E2 28668.173} C_VEL
LIN {X 0,Y 604.522,Z 350.064,A -85,B 0,C 180,E1 28667.928,E2 28667.928} C_VEL
LIN {X 0,Y 605.007,Z 354.037,A -85,B 0,C 180,E1 28667.585,E2 28667.585} C_VEL
LIN {X 0,Y 605.092,Z 356.363,A -85,B 0,C 180,E1 28667.195,E2 28667.195} C_VEL
LIN {X 0,Y 604.728,Z 357.353,A -85,B 0,C 180,E1 28666.672,E2 28666.672} C_VEL
LIN {X 0,Y 604.108,Z 356.595,A -85,B 0,C 180,E1 28666.188,E2 28666.188} C_VEL
LIN {X 0,Y 603.214,Z 353.672,A -85,B 0,C 180,E1 28665.594,E2 28665.594} C_VEL
LIN {X 0,Y 602.239,Z 348.152,A -85,B 0,C 180,E1 28664.945,E2 28664.945} C_VEL
LIN {X 0,Y 601.234,Z 339.228,A -85,B 0,C 180,E1 28664.212,E2 28664.212} C_VEL
LIN {X 0,Y 601.176,Z 285.293,A -85,B 0,C 180,E1 28660.382,E2 28660.382} C_VEL
LIN {X 0,Y 601.296,Z 248.823,A -85,B 0,C 180,E1 28657.672,E2 28657.672} C_VEL
LIN {X 0,Y 601.378,Z 241.621,A -85,B 0,C 180,E1 28657.123,E2 28657.123} C_VEL
LIN {X 0,Y 599.94,Z 238.004,A -85,B 0,C 180,E1 28656.7,E2 28656.7} C_VEL
LIN {X 0,Y 599.969,Z 238.002,A -85,B 0,C 180,E1 28653.564,E2 28653.564} C_VEL
LIN {X 0,Y 599.973,Z 238.003,A -85,B 0,C 180,E1 28650.316,E2 28650.316} C_VEL
LIN {X 0,Y 599.967,Z 237.999,A -85,B 0,C 180,E1 28647.062,E2 28647.062} C_VEL
LIN {X 0,Y 599.956,Z 238.158,A -85,B 0,C 180,E1 28646.195,E2 28646.195} C_VEL
LIN {X 0,Y 600.128,Z 266.247,A -85,B 0,C 180,E1 28644.405,E2 28644.405} C_VEL
LIN {X 0,Y 600.458,Z 294.301,A -85,B 0,C 180,E1 28642.519,E2 28642.519} C_VEL
LIN {X 0,Y 600.339,Z 337.592,A -85,B 0,C 180,E1 28639.406,E2 28639.406} C_VEL
LIN {X 0,Y 600.229,Z 381.769,A -85,B 0,C 180,E1 28636.301,E2 28636.301} C_VEL
LIN {X 0,Y 600.154,Z 427.523,A -85,B 0,C 180,E1 28633.147,E2 28633.147} C_VEL
LIN {X 0,Y 600.073,Z 476.428,A -85,B 0,C 180,E1 28629.833,E2 28629.833} C_VEL
LIN {X 0,Y 600.097,Z 486.074,A -85,B 0,C 180,E1 28629.211,E2 28629.211} C_VEL
LIN {X 0,Y 600.082,Z 599.901,A -85,B 0,C 180,E1 28627.819,E2 28627.819} C_VEL
LIN {X 0,Y 600.047,Z 614.466,A -85,B 0,C 180,E1 28627.468,E2 28627.468} C_VEL
LIN {X 0,Y 600.031,Z 628.726,A -85,B 0,C 180,E1 28626.939,E2 28626.939} C_VEL
LIN {X 0,Y 599.99,Z 641.905,A -85,B 0,C 180,E1 28626.266,E2 28626.266} C_VEL
LIN {X 0,Y 599.986,Z 654.787,A -85,B 0,C 180,E1 28625.402,E2 28625.402} C_VEL
LIN {X 0,Y 599.961,Z 666.372,A -85,B 0,C 180,E1 28624.396,E2 28624.396} C_VEL
LIN {X 0,Y 599.943,Z 675.957,A -85,B 0,C 180,E1 28623.344,E2 28623.344} C_VEL
LIN {X 0,Y 599.931,Z 684.205,A -85,B 0,C 180,E1 28622.196,E2 28622.196} C_VEL
LIN {X 0,Y 599.921,Z 691.521,A -85,B 0,C 180,E1 28620.859,E2 28620.859} C_VEL
LIN {X 0,Y 599.92,Z 696.79,A -85,B 0,C 180,E1 28619.522,E2 28619.522} C_VEL
LIN {X 0,Y 599.918,Z 700.492,A -85,B 0,C 180,E1 28618.089,E2 28618.089} C_VEL
LIN {X 0,Y 599.916,Z 702.33,A -85,B 0,C 180,E1 28616.56,E2 28616.56} C_VEL
LIN {X 0,Y 599.917,Z 702.174,A -85,B 0,C 180,E1 28615.124,E2 28615.124} C_VEL
LIN {X 0,Y 599.916,Z 700.203,A -85,B 0,C 180,E1 28613.684,E2 28613.684} C_VEL
LIN {X 0,Y 599.917,Z 699.685,A -85,B 0,C 180,E1 28613.441,E2 28613.441} C_VEL
LIN {X 0,Y 598.921,Z 697.904,A -85,B 0,C 180,E1 28612.725,E2 28612.725} C_VEL
LIN {X 0,Y 595.187,Z 694.31,A -85,B 0,C 180,E1 28611.653,E2 28611.653} C_VEL
LIN {X 0,Y 592.464,Z 690.572,A -85,B 0,C 180,E1 28610.787,E2 28610.787} C_VEL
LIN {X 0,Y 591.934,Z 688.117,A -85,B 0,C 180,E1 28610.304,E2 28610.304} C_VEL
LIN {X 0,Y 591.956,Z 680.663,A -85,B 0,C 180,E1 28609.095,E2 28609.095} C_VEL
LIN {X 0,Y 591.986,Z 671.237,A -85,B 0,C 180,E1 28607.91,E2 28607.91} C_VEL
LIN {X 0,Y 592.033,Z 660.154,A -85,B 0,C 180,E1 28606.821,E2 28606.821} C_VEL
LIN {X 0,Y 592.069,Z 648.482,A -85,B 0,C 180,E1 28605.925,E2 28605.925} C_VEL
LIN {X 0,Y 592.128,Z 636.071,A -85,B 0,C 180,E1 28605.177,E2 28605.177} C_VEL
LIN {X 0,Y 592.164,Z 622.104,A -85,B 0,C 180,E1 28604.552,E2 28604.552} C_VEL
LIN {X 0,Y 592.225,Z 607.683,A -85,B 0,C 180,E1 28604.098,E2 28604.098} C_VEL
LIN {X 0,Y 592.261,Z 592.1,A -85,B 0,C 180,E1 28603.812,E2 28603.812} C_VEL
LIN {X 0,Y 592.192,Z 485.55,A -85,B 0,C 180,E1 28602.51,E2 28602.51} C_VEL
LIN {X 0,Y 592.352,Z 438.518,A -85,B 0,C 180,E1 28599.29,E2 28599.29} C_VEL
LIN {X 0,Y 592.551,Z 391.977,A -85,B 0,C 180,E1 28596.053,E2 28596.053} C_VEL
LIN {X 0,Y 592.765,Z 345.275,A -85,B 0,C 180,E1 28592.74,E2 28592.74} C_VEL
LIN {X 0,Y 592.865,Z 306.212,A -85,B 0,C 180,E1 28589.941,E2 28589.941} C_VEL
LIN {X 0,Y 592.797,Z 258.858,A -85,B 0,C 180,E1 28586.578,E2 28586.578} C_VEL
LIN {X 0,Y 592.756,Z 241.795,A -85,B 0,C 180,E1 28585.403,E2 28585.403} C_VEL
LIN {X 0,Y 592,Z 238.995,A -85,B 0,C 180,E1 28585.169,E2 28585.169} C_VEL
LIN {X 0,Y 592.036,Z 238.987,A -85,B 0,C 180,E1 28581.944,E2 28581.944} C_VEL
LIN {X 0,Y 592.041,Z 238.992,A -85,B 0,C 180,E1 28578.577,E2 28578.577} C_VEL
LIN {X 0,Y 592.003,Z 238.993,A -85,B 0,C 180,E1 28575.321,E2 28575.321} C_VEL
LIN {X 0,Y 592.008,Z 238.992,A -85,B 0,C 180,E1 28572.237,E2 28572.237} C_VEL
LIN {X 0,Y 592.025,Z 238.993,A -85,B 0,C 180,E1 28568.923,E2 28568.923} C_VEL
LIN {X 0,Y 592.018,Z 239.135,A -85,B 0,C 180,E1 28566.691,E2 28566.691} C_VEL
LIN {X 0,Y 593.492,Z 244.4,A -85,B 0,C 180,E1 28566.132,E2 28566.132} C_VEL
LIN {X 0,Y 593.198,Z 281.057,A -85,B 0,C 180,E1 28562.986,E2 28562.986} C_VEL
LIN {X 0,Y 593.155,Z 300.759,A -85,B 0,C 180,E1 28561.364,E2 28561.364} C_VEL
LIN {X 0,Y 593.702,Z 304.896,A -85,B 0,C 180,E1 28561.28,E2 28561.28} C_VEL
LIN {X 0,Y 593.387,Z 535,A -85,B 0,C 180,E1 28558.239,E2 28558.239} C_VEL
LIN {X 0,Y 593.312,Z 564.137,A -85,B 0,C 180,E1 28557.812,E2 28557.812} C_VEL
LIN {X 0,Y 593.214,Z 584.344,A -85,B 0,C 180,E1 28557.341,E2 28557.341} C_VEL
LIN {X 0,Y 593.085,Z 604.422,A -85,B 0,C 180,E1 28556.682,E2 28556.682} C_VEL
LIN {X 0,Y 592.94,Z 623.867,A -85,B 0,C 180,E1 28555.857,E2 28555.857} C_VEL
LIN {X 0,Y 592.771,Z 643.226,A -85,B 0,C 180,E1 28554.835,E2 28554.835} C_VEL
LIN {X 0,Y 592.603,Z 661.401,A -85,B 0,C 180,E1 28553.676,E2 28553.676} C_VEL
LIN {X 0,Y 592.443,Z 678.753,A -85,B 0,C 180,E1 28552.352,E2 28552.352} C_VEL
LIN {X 0,Y 592.325,Z 694.223,A -85,B 0,C 180,E1 28550.969,E2 28550.969} C_VEL
LIN {X 0,Y 592.201,Z 708.883,A -85,B 0,C 180,E1 28549.428,E2 28549.428} C_VEL
LIN {X 0,Y 592.102,Z 722.472,A -85,B 0,C 180,E1 28547.747,E2 28547.747} C_VEL
LIN {X 0,Y 592.034,Z 734.522,A -85,B 0,C 180,E1 28545.979,E2 28545.979} C_VEL
LIN {X 0,Y 591.975,Z 744.742,A -85,B 0,C 180,E1 28544.177,E2 28544.177} C_VEL
LIN {X 0,Y 591.946,Z 753.563,A -85,B 0,C 180,E1 28542.288,E2 28542.288} C_VEL
LIN {X 0,Y 591.926,Z 760.543,A -85,B 0,C 180,E1 28540.413,E2 28540.413} C_VEL
LIN {X 0,Y 591.917,Z 766.078,A -85,B 0,C 180,E1 28538.451,E2 28538.451} C_VEL
LIN {X 0,Y 591.909,Z 769.97,A -85,B 0,C 180,E1 28536.401,E2 28536.401} C_VEL
LIN {X 0,Y 591.906,Z 771.973,A -85,B 0,C 180,E1 28534.457,E2 28534.457} C_VEL
LIN {X 0,Y 591.901,Z 772.389,A -85,B 0,C 180,E1 28532.42,E2 28532.42} C_VEL
LIN {X 0,Y 591.902,Z 771.061,A -85,B 0,C 180,E1 28530.387,E2 28530.387} C_VEL
LIN {X 0,Y 591.904,Z 768.185,A -85,B 0,C 180,E1 28528.451,E2 28528.451} C_VEL
LIN {X 0,Y 591.909,Z 763.631,A -85,B 0,C 180,E1 28526.514,E2 28526.514} C_VEL
LIN {X 0,Y 591.928,Z 757.659,A -85,B 0,C 180,E1 28524.669,E2 28524.669} C_VEL
LIN {X 0,Y 591.958,Z 749.597,A -85,B 0,C 180,E1 28522.722,E2 28522.722} C_VEL
LIN {X 0,Y 592.001,Z 740.068,A -85,B 0,C 180,E1 28520.865,E2 28520.865} C_VEL
LIN {X 0,Y 592.064,Z 729.116,A -85,B 0,C 180,E1 28519.097,E2 28519.097} C_VEL
LIN {X 0,Y 592.14,Z 716.721,A -85,B 0,C 180,E1 28517.419,E2 28517.419} C_VEL
LIN {X 0,Y 592.24,Z 702.941,A -85,B 0,C 180,E1 28515.83,E2 28515.83} C_VEL
LIN {X 0,Y 592.366,Z 687.683,A -85,B 0,C 180,E1 28514.332,E2 28514.332} C_VEL
LIN {X 0,Y 592.516,Z 671.195,A -85,B 0,C 180,E1 28512.953,E2 28512.953} C_VEL
LIN {X 0,Y 592.678,Z 653.604,A -85,B 0,C 180,E1 28511.712,E2 28511.712} C_VEL
LIN {X 0,Y 592.849,Z 635.625,A -85,B 0,C 180,E1 28510.646,E2 28510.646} C_VEL
LIN {X 0,Y 593.002,Z 616.751,A -85,B 0,C 180,E1 28509.727,E2 28509.727} C_VEL
LIN {X 0,Y 593.124,Z 597.535,A -85,B 0,C 180,E1 28508.983,E2 28508.983} C_VEL
LIN {X 0,Y 593.243,Z 577.25,A -85,B 0,C 180,E1 28508.385,E2 28508.385} C_VEL
LIN {X 0,Y 593.344,Z 556.431,A -85,B 0,C 180,E1 28507.965,E2 28507.965} C_VEL
LIN {X 0,Y 593.737,Z 306.894,A -85,B 0,C 180,E1 28504.659,E2 28504.659} C_VEL
LIN {X 0,Y 593.471,Z 300.626,A -85,B 0,C 180,E1 28504.561,E2 28504.561} C_VEL
LIN {X 0,Y 593.223,Z 298.755,A -85,B 0,C 180,E1 28504.492,E2 28504.492} C_VEL
LIN {X 0,Y 593.492,Z 254.646,A -85,B 0,C 180,E1 28501.305,E2 28501.305} C_VEL
LIN {X 0,Y 593.455,Z 243.394,A -85,B 0,C 180,E1 28500.469,E2 28500.469} C_VEL
LIN {X 0,Y 592.035,Z 238.993,A -85,B 0,C 180,E1 28500.042,E2 28500.042} C_VEL
LIN {X 0,Y 592.017,Z 238.993,A -85,B 0,C 180,E1 28496.824,E2 28496.824} C_VEL
LIN {X 0,Y 592.011,Z 238.994,A -85,B 0,C 180,E1 28493.643,E2 28493.643} C_VEL
LIN {X 0,Y 592.04,Z 238.993,A -85,B 0,C 180,E1 28490.454,E2 28490.454} C_VEL
LIN {X 0,Y 592.028,Z 238.993,A -85,B 0,C 180,E1 28487.108,E2 28487.108} C_VEL
LIN {X 0,Y 592.027,Z 238.991,A -85,B 0,C 180,E1 28483.824,E2 28483.824} C_VEL
LIN {X 0,Y 592.026,Z 238.989,A -85,B 0,C 180,E1 28480.684,E2 28480.684} C_VEL
LIN {X 0,Y 592.035,Z 238.99,A -85,B 0,C 180,E1 28477.445,E2 28477.445} C_VEL
LIN {X 0,Y 592.037,Z 238.991,A -85,B 0,C 180,E1 28474.104,E2 28474.104} C_VEL
LIN {X 0,Y 592.01,Z 238.993,A -85,B 0,C 180,E1 28470.893,E2 28470.893} C_VEL
LIN {X 0,Y 592.026,Z 238.993,A -85,B 0,C 180,E1 28467.751,E2 28467.751} C_VEL
LIN {X 0,Y 592.038,Z 239.071,A -85,B 0,C 180,E1 28466.262,E2 28466.262} C_VEL
LIN {X 0,Y 592.797,Z 242.449,A -85,B 0,C 180,E1 28465.972,E2 28465.972} C_VEL
LIN {X 0,Y 592.916,Z 286.421,A -85,B 0,C 180,E1 28462.612,E2 28462.612} C_VEL
LIN {X 0,Y 592.871,Z 318.555,A -85,B 0,C 180,E1 28460.124,E2 28460.124} C_VEL
LIN {X 0,Y 592.638,Z 360.704,A -85,B 0,C 180,E1 28456.87,E2 28456.87} C_VEL
LIN {X 0,Y 592.439,Z 404.51,A -85,B 0,C 180,E1 28453.56,E2 28453.56} C_VEL
LIN {X 0,Y 592.351,Z 436.447,A -85,B 0,C 180,E1 28451.211,E2 28451.211} C_VEL
LIN {X 0,Y 592.386,Z 578.876,A -85,B 0,C 180,E1 28449.429,E2 28449.429} C_VEL
LIN {X 0,Y 592.344,Z 596.244,A -85,B 0,C 180,E1 28449.008,E2 28449.008} C_VEL
LIN {X 0,Y 592.272,Z 611.613,A -85,B 0,C 180,E1 28448.446,E2 28448.446} C_VEL
LIN {X 0,Y 592.203,Z 627.434,A -85,B 0,C 180,E1 28447.657,E2 28447.657} C_VEL
LIN {X 0,Y 592.136,Z 640.865,A -85,B 0,C 180,E1 28446.789,E2 28446.789} C_VEL
LIN {X 0,Y 592.07,Z 654.618,A -85,B 0,C 180,E1 28445.67,E2 28445.67} C_VEL
LIN {X 0,Y 592.011,Z 665.559,A -85,B 0,C 180,E1 28444.553,E2 28444.553} C_VEL
LIN {X 0,Y 591.974,Z 675.587,A -85,B 0,C 180,E1 28443.292,E2 28443.292} C_VEL
LIN {X 0,Y 591.945,Z 684.172,A -85,B 0,C 180,E1 28441.936,E2 28441.936} C_VEL
LIN {X 0,Y 591.929,Z 691.238,A -85,B 0,C 180,E1 28440.484,E2 28440.484} C_VEL
LIN {X 0,Y 591.917,Z 696.772,A -85,B 0,C 180,E1 28438.936,E2 28438.936} C_VEL
LIN {X 0,Y 591.916,Z 700.359,A -85,B 0,C 180,E1 28437.386,E2 28437.386} C_VEL
LIN {X 0,Y 591.914,Z 702.263,A -85,B 0,C 180,E1 28435.738,E2 28435.738} C_VEL
LIN {X 0,Y 591.914,Z 702.259,A -85,B 0,C 180,E1 28434.183,E2 28434.183} C_VEL
LIN {X 0,Y 591.913,Z 700.523,A -85,B 0,C 180,E1 28432.624,E2 28432.624} C_VEL
LIN {X 0,Y 591.917,Z 697.027,A -85,B 0,C 180,E1 28431.06,E2 28431.06} C_VEL
LIN {X 0,Y 591.924,Z 691.897,A -85,B 0,C 180,E1 28429.587,E2 28429.587} C_VEL
LIN {X 0,Y 591.941,Z 684.901,A -85,B 0,C 180,E1 28428.108,E2 28428.108} C_VEL
LIN {X 0,Y 591.971,Z 676.312,A -85,B 0,C 180,E1 28426.72,E2 28426.72} C_VEL
LIN {X 0,Y 592.01,Z 666.041,A -85,B 0,C 180,E1 28425.412,E2 28425.412} C_VEL
LIN {X 0,Y 592.069,Z 654.422,A -85,B 0,C 180,E1 28424.224,E2 28424.224} C_VEL
LIN {X 0,Y 592.129,Z 641.471,A -85,B 0,C 180,E1 28423.167,E2 28423.167} C_VEL
LIN {X 0,Y 592.195,Z 628.401,A -85,B 0,C 180,E1 28422.308,E2 28422.308} C_VEL
LIN {X 0,Y 592.263,Z 613.462,A -85,B 0,C 180,E1 28421.547,E2 28421.547} C_VEL
LIN {X 0,Y 592.338,Z 598.046,A -85,B 0,C 180,E1 28420.958,E2 28420.958} C_VEL
LIN {X 0,Y 592.386,Z 581.855,A -85,B 0,C 180,E1 28420.538,E2 28420.538} C_VEL
LIN {X 0,Y 592.42,Z 558.26,A -85,B 0,C 180,E1 28420.202,E2 28420.202} C_VEL
LIN {X 0,Y 592.318,Z 436.016,A -85,B 0,C 180,E1 28418.692,E2 28418.692} C_VEL
LIN {X 0,Y 592.482,Z 392.81,A -85,B 0,C 180,E1 28415.472,E2 28415.472} C_VEL
LIN {X 0,Y 592.702,Z 349.678,A -85,B 0,C 180,E1 28412.197,E2 28412.197} C_VEL
LIN {X 0,Y 592.928,Z 308.348,A -85,B 0,C 180,E1 28408.986,E2 28408.986} C_VEL
LIN {X 0,Y 592.825,Z 288.032,A -85,B 0,C 180,E1 28407.451,E2 28407.451} C_VEL
LIN {X 0,Y 592.357,Z 263.839,A -85,B 0,C 180,E1 28405.748,E2 28405.748} C_VEL
LIN {X 0,Y 592.019,Z 238.993,A -85,B 0,C 180,E1 28404.093,E2 28404.093} C_VEL
LIN {X 0,Y 592.039,Z 238.989,A -85,B 0,C 180,E1 28400.822,E2 28400.822} C_VEL
LIN {X 0,Y 592.054,Z 239.125,A -85,B 0,C 180,E1 28400.344,E2 28400.344} C_VEL
LIN {X 0,Y 593.172,Z 242.233,A -85,B 0,C 180,E1 28400.043,E2 28400.043} C_VEL
LIN {X 0,Y 594.867,Z 245.891,A -85,B 0,C 180,E1 28399.66,E2 28399.66} C_VEL
LIN {X 0,Y 594.818,Z 304.262,A -85,B 0,C 180,E1 28395.967,E2 28395.967} C_VEL
LIN {X 0,Y 596.484,Z 315.515,A -85,B 0,C 180,E1 28395.159,E2 28395.159} C_VEL
LIN {X 0,Y 598.484,Z 322.042,A -85,B 0,C 180,E1 28394.562,E2 28394.562} C_VEL
LIN {X 0,Y 600.337,Z 325.817,A -85,B 0,C 180,E1 28393.988,E2 28393.988} C_VEL
LIN {X 0,Y 601.779,Z 327.429,A -85,B 0,C 180,E1 28393.442,E2 28393.442} C_VEL
LIN {X 0,Y 602.61,Z 327.433,A -85,B 0,C 180,E1 28392.97,E2 28392.97} C_VEL
LIN {X 0,Y 602.919,Z 325.841,A -85,B 0,C 180,E1 28392.441,E2 28392.441} C_VEL
LIN {X 0,Y 602.435,Z 322.708,A -85,B 0,C 180,E1 28391.979,E2 28391.979} C_VEL
LIN {X 0,Y 601.209,Z 318.132,A -85,B 0,C 180,E1 28391.605,E2 28391.605} C_VEL
LIN {X 0,Y 599.437,Z 311.902,A -85,B 0,C 180,E1 28391.348,E2 28391.348} C_VEL
LIN {X 0,Y 597.85,Z 302.688,A -85,B 0,C 180,E1 28391.175,E2 28391.175} C_VEL
LIN {X 0,Y 597.254,Z 290.599,A -85,B 0,C 180,E1 28391.11,E2 28391.11} C_VEL
LIN {X 0,Y 597.089,Z 246.423,A -85,B 0,C 180,E1 28391.092,E2 28391.092} C_VEL
LIN {X 0,Y 596.105,Z 245.007,A -85,B 0,C 180,E1 28390.983,E2 28390.983} C_VEL
LIN {X 0,Y 593.407,Z 242.56,A -85,B 0,C 180,E1 28390.683,E2 28390.683} C_VEL
LIN {X 0,Y 592.11,Z 239.464,A -85,B 0,C 180,E1 28390.536,E2 28390.536} C_VEL
LIN {X 0,Y 592.036,Z 238.99,A -85,B 0,C 180,E1 28390.517,E2 28390.517} C_VEL
LIN {X 0,Y 592.049,Z 239.108,A -85,B 0,C 180,E1 28387.2,E2 28387.2} C_VEL
LIN {X 0,Y 593.029,Z 241.974,A -85,B 0,C 180,E1 28386.949,E2 28386.949} C_VEL
LIN {X 0,Y 594.304,Z 244.918,A -85,B 0,C 180,E1 28386.674,E2 28386.674} C_VEL
LIN {X 0,Y 593.948,Z 295.279,A -85,B 0,C 180,E1 28383.631,E2 28383.631} C_VEL
LIN {X 0,Y 594.02,Z 302.684,A -85,B 0,C 180,E1 28383.216,E2 28383.216} C_VEL
LIN {X 0,Y 594.41,Z 307.324,A -85,B 0,C 180,E1 28383.126,E2 28383.126} C_VEL
LIN {X 0,Y 593.973,Z 527.634,A -85,B 0,C 180,E1 28380.089,E2 28380.089} C_VEL
LIN {X 0,Y 593.812,Z 608.964,A -85,B 0,C 180,E1 28378.96,E2 28378.96} C_VEL
LIN {X 0,Y 593.692,Z 630.429,A -85,B 0,C 180,E1 28378.475,E2 28378.475} C_VEL
LIN {X 0,Y 593.516,Z 652.521,A -85,B 0,C 180,E1 28377.79,E2 28377.79} C_VEL
LIN {X 0,Y 593.367,Z 673.438,A -85,B 0,C 180,E1 28376.951,E2 28376.951} C_VEL
LIN {X 0,Y 593.173,Z 692.746,A -85,B 0,C 180,E1 28375.993,E2 28375.993} C_VEL
LIN {X 0,Y 592.956,Z 712.535,A -85,B 0,C 180,E1 28374.827,E2 28374.827} C_VEL
LIN {X 0,Y 592.781,Z 731.694,A -85,B 0,C 180,E1 28373.491,E2 28373.491} C_VEL
LIN {X 0,Y 592.583,Z 750.232,A -85,B 0,C 180,E1 28371.97,E2 28371.97} C_VEL
LIN {X 0,Y 592.409,Z 767.205,A -85,B 0,C 180,E1 28370.346,E2 28370.346} C_VEL
LIN {X 0,Y 592.26,Z 782.871,A -85,B 0,C 180,E1 28368.607,E2 28368.607} C_VEL
LIN {X 0,Y 592.135,Z 797.05,A -85,B 0,C 180,E1 28366.782,E2 28366.782} C_VEL
LIN {X 0,Y 592.056,Z 809.745,A -85,B 0,C 180,E1 28364.874,E2 28364.874} C_VEL
LIN {X 0,Y 591.988,Z 820.463,A -85,B 0,C 180,E1 28362.957,E2 28362.957} C_VEL
LIN {X 0,Y 591.943,Z 830.072,A -85,B 0,C 180,E1 28360.905,E2 28360.905} C_VEL
LIN {X 0,Y 591.935,Z 837.598,A -85,B 0,C 180,E1 28358.94,E2 28358.94} C_VEL
LIN {X 0,Y 591.924,Z 843.659,A -85,B 0,C 180,E1 28356.888,E2 28356.888} C_VEL
LIN {X 0,Y 591.914,Z 848.369,A -85,B 0,C 180,E1 28354.711,E2 28354.711} C_VEL
LIN {X 0,Y 591.905,Z 851.238,A -85,B 0,C 180,E1 28352.614,E2 28352.614} C_VEL
LIN {X 0,Y 591.897,Z 852.379,A -85,B 0,C 180,E1 28350.581,E2 28350.581} C_VEL
LIN {X 0,Y 591.897,Z 852.019,A -85,B 0,C 180,E1 28348.451,E2 28348.451} C_VEL
LIN {X 0,Y 591.902,Z 850.116,A -85,B 0,C 180,E1 28346.417,E2 28346.417} C_VEL
LIN {X 0,Y 591.918,Z 846.608,A -85,B 0,C 180,E1 28344.377,E2 28344.377} C_VEL
LIN {X 0,Y 591.922,Z 841.587,A -85,B 0,C 180,E1 28342.331,E2 28342.331} C_VEL
LIN {X 0,Y 591.929,Z 834.759,A -85,B 0,C 180,E1 28340.275,E2 28340.275} C_VEL
LIN {X 0,Y 591.96,Z 826.142,A -85,B 0,C 180,E1 28338.207,E2 28338.207} C_VEL
LIN {X 0,Y 592.013,Z 816.132,A -85,B 0,C 180,E1 28336.223,E2 28336.223} C_VEL
LIN {X 0,Y 592.085,Z 804.294,A -85,B 0,C 180,E1 28334.272,E2 28334.272} C_VEL
LIN {X 0,Y 592.192,Z 791.014,A -85,B 0,C 180,E1 28332.409,E2 28332.409} C_VEL
LIN {X 0,Y 592.324,Z 775.815,A -85,B 0,C 180,E1 28330.577,E2 28330.577} C_VEL
LIN {X 0,Y 592.486,Z 760.009,A -85,B 0,C 180,E1 28328.933,E2 28328.933} C_VEL
LIN {X 0,Y 592.667,Z 742.204,A -85,B 0,C 180,E1 28327.341,E2 28327.341} C_VEL
LIN {X 0,Y 592.841,Z 723.476,A -85,B 0,C 180,E1 28325.911,E2 28325.911} C_VEL
LIN {X 0,Y 593.056,Z 703.954,A -85,B 0,C 180,E1 28324.644,E2 28324.644} C_VEL
LIN {X 0,Y 593.26,Z 684.626,A -85,B 0,C 180,E1 28323.58,E2 28323.58} C_VEL
LIN {X 0,Y 593.424,Z 664.507,A -85,B 0,C 180,E1 28322.668,E2 28322.668} C_VEL
LIN {X 0,Y 593.611,Z 643.271,A -85,B 0,C 180,E1 28321.901,E2 28321.901} C_VEL
LIN {X 0,Y 593.744,Z 622.042,A -85,B 0,C 180,E1 28321.312,E2 28321.312} C_VEL
LIN {X 0,Y 593.842,Z 600.539,A -85,B 0,C 180,E1 28320.905,E2 28320.905} C_VEL
LIN {X 0,Y 594.249,Z 371.105,A -85,B 0,C 180,E1 28317.761,E2 28317.761} C_VEL
LIN {X 0,Y 594.229,Z 305.139,A -85,B 0,C 180,E1 28316.831,E2 28316.831} C_VEL
LIN {X 0,Y 593.747,Z 302.732,A -85,B 0,C 180,E1 28316.76,E2 28316.76} C_VEL
LIN {X 0,Y 594.05,Z 259.684,A -85,B 0,C 180,E1 28313.727,E2 28313.727} C_VEL
LIN {X 0,Y 594.102,Z 244.67,A -85,B 0,C 180,E1 28312.639,E2 28312.639} C_VEL
LIN {X 0,Y 592.036,Z 238.993,A -85,B 0,C 180,E1 28312.063,E2 28312.063} C_VEL
LIN {X 0,Y 592.059,Z 239.154,A -85,B 0,C 180,E1 28309.47,E2 28309.47} C_VEL
LIN {X 0,Y 593.164,Z 242.191,A -85,B 0,C 180,E1 28309.345,E2 28309.345} C_VEL
LIN {X 0,Y 595.613,Z 244.719,A -85,B 0,C 180,E1 28309.071,E2 28309.071} C_VEL
LIN {X 0,Y 596.679,Z 245.709,A -85,B 0,C 180,E1 28308.953,E2 28308.953} C_VEL
LIN {X 0,Y 597.259,Z 246.727,A -85,B 0,C 180,E1 28308.889,E2 28308.889} C_VEL
LIN {X 0,Y 597.439,Z 335.781,A -85,B 0,C 180,E1 28308.87,E2 28308.87} C_VEL
LIN {X 0,Y 598.571,Z 345.755,A -85,B 0,C 180,E1 28308.746,E2 28308.746} C_VEL
LIN {X 0,Y 600.391,Z 353.143,A -85,B 0,C 180,E1 28308.52,E2 28308.52} C_VEL
LIN {X 0,Y 601.654,Z 358.139,A -85,B 0,C 180,E1 28308.194,E2 28308.194} C_VEL
LIN {X 0,Y 602.272,Z 361.874,A -85,B 0,C 180,E1 28307.75,E2 28307.75} C_VEL
LIN {X 0,Y 602.221,Z 363.688,A -85,B 0,C 180,E1 28307.35,E2 28307.35} C_VEL
LIN {X 0,Y 601.586,Z 364.565,A -85,B 0,C 180,E1 28306.855,E2 28306.855} C_VEL
LIN {X 0,Y 600.255,Z 363.839,A -85,B 0,C 180,E1 28306.268,E2 28306.268} C_VEL
LIN {X 0,Y 598.676,Z 361.404,A -85,B 0,C 180,E1 28305.724,E2 28305.724} C_VEL
LIN {X 0,Y 596.809,Z 356.572,A -85,B 0,C 180,E1 28305.126,E2 28305.126} C_VEL
LIN {X 0,Y 594.751,Z 346.873,A -85,B 0,C 180,E1 28304.307,E2 28304.307} C_VEL
LIN {X 0,Y 594.073,Z 331.447,A -85,B 0,C 180,E1 28303.176,E2 28303.176} C_VEL
LIN {X 0,Y 594.441,Z 289.526,A -85,B 0,C 180,E1 28300.169,E2 28300.169} C_VEL
LIN {X 0,Y 594.741,Z 253.783,A -85,B 0,C 180,E1 28297.484,E2 28297.484} C_VEL
LIN {X 0,Y 594.765,Z 245.696,A -85,B 0,C 180,E1 28296.85,E2 28296.85} C_VEL
LIN {X 0,Y 592.062,Z 239.418,A -85,B 0,C 180,E1 28296.096,E2 28296.096} C_VEL
LIN {X 0,Y 592.005,Z 238.997,A -85,B 0,C 180,E1 28295.997,E2 28295.997} C_VEL
LIN {X 0,Y 592.021,Z 238.989,A -85,B 0,C 180,E1 28292.714,E2 28292.714} C_VEL
LIN {X 0,Y 592.009,Z 238.99,A -85,B 0,C 180,E1 28289.549,E2 28289.549} C_VEL
LIN {X 0,Y 592.035,Z 239.186,A -85,B 0,C 180,E1 28286.325,E2 28286.325} C_VEL
LIN {X 0,Y 592.428,Z 276.712,A -85,B 0,C 180,E1 28283.932,E2 28283.932} C_VEL
LIN {X 0,Y 592.898,Z 318.493,A -85,B 0,C 180,E1 28281.103,E2 28281.103} C_VEL
LIN {X 0,Y 592.677,Z 363.33,A -85,B 0,C 180,E1 28277.88,E2 28277.88} C_VEL
LIN {X 0,Y 592.466,Z 410.474,A -85,B 0,C 180,E1 28274.563,E2 28274.563} C_VEL
LIN {X 0,Y 592.297,Z 457.822,A -85,B 0,C 180,E1 28271.292,E2 28271.292} C_VEL
LIN {X 0,Y 592.249,Z 486.127,A -85,B 0,C 180,E1 28269.39,E2 28269.39} C_VEL
LIN {X 0,Y 592.25,Z 600.088,A -85,B 0,C 180,E1 28267.975,E2 28267.975} C_VEL
LIN {X 0,Y 592.195,Z 614.945,A -85,B 0,C 180,E1 28267.607,E2 28267.607} C_VEL
LIN {X 0,Y 592.154,Z 629.957,A -85,B 0,C 180,E1 28267.031,E2 28267.031} C_VEL
LIN {X 0,Y 592.083,Z 642.81,A -85,B 0,C 180,E1 28266.35,E2 28266.35} C_VEL
LIN {X 0,Y 592.051,Z 655.469,A -85,B 0,C 180,E1 28265.475,E2 28265.475} C_VEL
LIN {X 0,Y 592.004,Z 666.926,A -85,B 0,C 180,E1 28264.456,E2 28264.456} C_VEL
LIN {X 0,Y 591.966,Z 677.165,A -85,B 0,C 180,E1 28263.292,E2 28263.292} C_VEL
LIN {X 0,Y 591.941,Z 685.125,A -85,B 0,C 180,E1 28262.129,E2 28262.129} C_VEL
LIN {X 0,Y 591.925,Z 692.226,A -85,B 0,C 180,E1 28260.774,E2 28260.774} C_VEL
LIN {X 0,Y 591.921,Z 697.255,A -85,B 0,C 180,E1 28259.419,E2 28259.419} C_VEL
LIN {X 0,Y 591.918,Z 700.594,A -85,B 0,C 180,E1 28258.064,E2 28258.064} C_VEL
LIN {X 0,Y 591.917,Z 702.346,A -85,B 0,C 180,E1 28256.513,E2 28256.513} C_VEL
LIN {X 0,Y 591.915,Z 702.137,A -85,B 0,C 180,E1 28255.058,E2 28255.058} C_VEL
LIN {X 0,Y 591.916,Z 700.083,A -85,B 0,C 180,E1 28253.599,E2 28253.599} C_VEL
LIN {X 0,Y 591.92,Z 696.454,A -85,B 0,C 180,E1 28252.233,E2 28252.233} C_VEL
LIN {X 0,Y 591.927,Z 690.951,A -85,B 0,C 180,E1 28250.863,E2 28250.863} C_VEL
LIN {X 0,Y 591.934,Z 688.117,A -85,B 0,C 180,E1 28250.304,E2 28250.304} C_VEL
LIN {X 0,Y 590.948,Z 684.437,A -85,B 0,C 180,E1 28249.649,E2 28249.649} C_VEL
LIN {X 0,Y 586.879,Z 677.55,A -85,B 0,C 180,E1 28248.598,E2 28248.598} C_VEL
LIN {X 0,Y 584.371,Z 671.589,A -85,B 0,C 180,E1 28247.843,E2 28247.843} C_VEL
LIN {X 0,Y 584.04,Z 668.656,A -85,B 0,C 180,E1 28247.516,E2 28247.516} C_VEL
LIN {X 0,Y 584.103,Z 658.269,A -85,B 0,C 180,E1 28246.537,E2 28246.537} C_VEL
LIN {X 0,Y 584.165,Z 646.165,A -85,B 0,C 180,E1 28245.63,E2 28245.63} C_VEL
LIN {X 0,Y 584.259,Z 632.823,A -85,B 0,C 180,E1 28244.866,E2 28244.866} C_VEL
LIN {X 0,Y 584.324,Z 619.233,A -85,B 0,C 180,E1 28244.288,E2 28244.288} C_VEL
LIN {X 0,Y 584.409,Z 603.338,A -85,B 0,C 180,E1 28243.836,E2 28243.836} C_VEL
LIN {X 0,Y 584.443,Z 584.57,A -85,B 0,C 180,E1 28243.554,E2 28243.554} C_VEL
LIN {X 0,Y 584.347,Z 485.432,A -85,B 0,C 180,E1 28242.318,E2 28242.318} C_VEL
LIN {X 0,Y 584.581,Z 439.159,A -85,B 0,C 180,E1 28239.107,E2 28239.107} C_VEL
LIN {X 0,Y 584.881,Z 392.472,A -85,B 0,C 180,E1 28235.816,E2 28235.816} C_VEL
LIN {X 0,Y 585.2,Z 346.699,A -85,B 0,C 180,E1 28232.528,E2 28232.528} C_VEL
LIN {X 0,Y 585.233,Z 313.685,A -85,B 0,C 180,E1 28230.187,E2 28230.187} C_VEL
LIN {X 0,Y 585.232,Z 267.014,A -85,B 0,C 180,E1 28226.842,E2 28226.842} C_VEL
LIN {X 0,Y 585.254,Z 244.301,A -85,B 0,C 180,E1 28225.261,E2 28225.261} C_VEL
LIN {X 0,Y 584.059,Z 239.984,A -85,B 0,C 180,E1 28224.886,E2 28224.886} C_VEL
LIN {X 0,Y 584.1,Z 239.978,A -85,B 0,C 180,E1 28221.582,E2 28221.582} C_VEL
LIN {X 0,Y 584.09,Z 239.98,A -85,B 0,C 180,E1 28218.276,E2 28218.276} C_VEL
LIN {X 0,Y 584.061,Z 239.983,A -85,B 0,C 180,E1 28214.855,E2 28214.855} C_VEL
LIN {X 0,Y 584.098,Z 239.981,A -85,B 0,C 180,E1 28211.62,E2 28211.62} C_VEL
LIN {X 0,Y 584.083,Z 239.981,A -85,B 0,C 180,E1 28208.369,E2 28208.369} C_VEL
LIN {X 0,Y 584.088,Z 239.988,A -85,B 0,C 180,E1 28207.135,E2 28207.135} C_VEL
LIN {X 0,Y 586.29,Z 247.131,A -85,B 0,C 180,E1 28206.35,E2 28206.35} C_VEL
LIN {X 0,Y 585.854,Z 283.854,A -85,B 0,C 180,E1 28203.161,E2 28203.161} C_VEL
LIN {X 0,Y 585.781,Z 300.703,A -85,B 0,C 180,E1 28201.756,E2 28201.756} C_VEL
LIN {X 0,Y 586.656,Z 306.042,A -85,B 0,C 180,E1 28201.636,E2 28201.636} C_VEL
LIN {X 0,Y 586.149,Z 536.73,A -85,B 0,C 180,E1 28198.551,E2 28198.551} C_VEL
LIN {X 0,Y 586.035,Z 564.73,A -85,B 0,C 180,E1 28198.13,E2 28198.13} C_VEL
LIN {X 0,Y 585.886,Z 584.835,A -85,B 0,C 180,E1 28197.651,E2 28197.651} C_VEL
LIN {X 0,Y 585.695,Z 604.81,A -85,B 0,C 180,E1 28196.984,E2 28196.984} C_VEL
LIN {X 0,Y 585.483,Z 623.214,A -85,B 0,C 180,E1 28196.197,E2 28196.197} C_VEL
LIN {X 0,Y 585.225,Z 642.462,A -85,B 0,C 180,E1 28195.177,E2 28195.177} C_VEL
LIN {X 0,Y 585.004,Z 660.044,A -85,B 0,C 180,E1 28194.056,E2 28194.056} C_VEL
LIN {X 0,Y 584.758,Z 677.837,A -85,B 0,C 180,E1 28192.696,E2 28192.696} C_VEL
LIN {X 0,Y 584.551,Z 693.77,A -85,B 0,C 180,E1 28191.261,E2 28191.261} C_VEL
LIN {X 0,Y 584.352,Z 709.382,A -85,B 0,C 180,E1 28189.595,E2 28189.595} C_VEL
LIN {X 0,Y 584.203,Z 722.86,A -85,B 0,C 180,E1 28187.899,E2 28187.899} C_VEL
LIN {X 0,Y 584.096,Z 734.901,A -85,B 0,C 180,E1 28186.1,E2 28186.1} C_VEL
LIN {X 0,Y 584.011,Z 745.045,A -85,B 0,C 180,E1 28184.273,E2 28184.273} C_VEL
LIN {X 0,Y 583.962,Z 753.806,A -85,B 0,C 180,E1 28182.358,E2 28182.358} C_VEL
LIN {X 0,Y 583.932,Z 761.028,A -85,B 0,C 180,E1 28180.358,E2 28180.358} C_VEL
LIN {X 0,Y 583.918,Z 766.421,A -85,B 0,C 180,E1 28178.369,E2 28178.369} C_VEL
LIN {X 0,Y 583.91,Z 770.059,A -85,B 0,C 180,E1 28176.391,E2 28176.391} C_VEL
LIN {X 0,Y 583.906,Z 772.013,A -85,B 0,C 180,E1 28174.419,E2 28174.419} C_VEL
LIN {X 0,Y 583.902,Z 772.378,A -85,B 0,C 180,E1 28172.355,E2 28172.355} C_VEL
LIN {X 0,Y 583.906,Z 770.997,A -85,B 0,C 180,E1 28170.294,E2 28170.294} C_VEL
LIN {X 0,Y 583.914,Z 767.862,A -85,B 0,C 180,E1 28168.234,E2 28168.234} C_VEL
LIN {X 0,Y 583.925,Z 763.196,A -85,B 0,C 180,E1 28166.269,E2 28166.269} C_VEL
LIN {X 0,Y 583.948,Z 756.752,A -85,B 0,C 180,E1 28164.301,E2 28164.301} C_VEL
LIN {X 0,Y 583.981,Z 748.874,A -85,B 0,C 180,E1 28162.424,E2 28162.424} C_VEL
LIN {X 0,Y 584.049,Z 739.169,A -85,B 0,C 180,E1 28160.541,E2 28160.541} C_VEL
LIN {X 0,Y 584.146,Z 728.011,A -85,B 0,C 180,E1 28158.748,E2 28158.748} C_VEL
LIN {X 0,Y 584.286,Z 715.474,A -85,B 0,C 180,E1 28157.046,E2 28157.046} C_VEL
LIN {X 0,Y 584.465,Z 700.509,A -85,B 0,C 180,E1 28155.334,E2 28155.334} C_VEL
LIN {X 0,Y 584.67,Z 684.834,A -85,B 0,C 180,E1 28153.814,E2 28153.814} C_VEL
LIN {X 0,Y 584.909,Z 667.429,A -85,B 0,C 180,E1 28152.388,E2 28152.388} C_VEL
LIN {X 0,Y 585.131,Z 650.226,A -85,B 0,C 180,E1 28151.204,E2 28151.204} C_VEL
LIN {X 0,Y 585.363,Z 631.578,A -85,B 0,C 180,E1 28150.128,E2 28150.128} C_VEL
LIN {X 0,Y 585.597,Z 612.856,A -85,B 0,C 180,E1 28149.25,E2 28149.25} C_VEL
LIN {X 0,Y 585.823,Z 592.985,A -85,B 0,C 180,E1 28148.508,E2 28148.508} C_VEL
LIN {X 0,Y 585.979,Z 572.553,A -85,B 0,C 180,E1 28147.944,E2 28147.944} C_VEL
LIN {X 0,Y 586.095,Z 552.546,A -85,B 0,C 180,E1 28147.573,E2 28147.573} C_VEL
LIN {X 0,Y 586.674,Z 311.17,A -85,B 0,C 180,E1 28144.345,E2 28144.345} C_VEL
LIN {X 0,Y 586.45,Z 302.093,A -85,B 0,C 180,E1 28144.209,E2 28144.209} C_VEL
LIN {X 0,Y 585.909,Z 299.024,A -85,B 0,C 180,E1 28144.123,E2 28144.123} C_VEL
LIN {X 0,Y 586.351,Z 253.802,A -85,B 0,C 180,E1 28140.811,E2 28140.811} C_VEL
LIN {X 0,Y 586.275,Z 246.237,A -85,B 0,C 180,E1 28140.236,E2 28140.236} C_VEL
LIN {X 0,Y 584.073,Z 239.983,A -85,B 0,C 180,E1 28139.592,E2 28139.592} C_VEL
LIN {X 0,Y 584.091,Z 239.982,A -85,B 0,C 180,E1 28136.314,E2 28136.314} C_VEL
LIN {X 0,Y 584.088,Z 239.984,A -85,B 0,C 180,E1 28133.069,E2 28133.069} C_VEL
LIN {X 0,Y 584.083,Z 239.982,A -85,B 0,C 180,E1 28129.773,E2 28129.773} C_VEL
LIN {X 0,Y 584.092,Z 239.979,A -85,B 0,C 180,E1 28126.516,E2 28126.516} C_VEL
LIN {X 0,Y 584.086,Z 239.982,A -85,B 0,C 180,E1 28123.215,E2 28123.215} C_VEL
LIN {X 0,Y 584.098,Z 239.98,A -85,B 0,C 180,E1 28119.808,E2 28119.808} C_VEL
LIN {X 0,Y 584.08,Z 239.978,A -85,B 0,C 180,E1 28116.565,E2 28116.565} C_VEL
LIN {X 0,Y 584.072,Z 239.982,A -85,B 0,C 180,E1 28113.342,E2 28113.342} C_VEL
LIN {X 0,Y 584.102,Z 239.98,A -85,B 0,C 180,E1 28110.103,E2 28110.103} C_VEL
LIN {X 0,Y 584.097,Z 239.982,A -85,B 0,C 180,E1 28106.647,E2 28106.647} C_VEL
LIN {X 0,Y 584.112,Z 240.131,A -85,B 0,C 180,E1 28106.537,E2 28106.537} C_VEL
LIN {X 0,Y 585.252,Z 245.142,A -85,B 0,C 180,E1 28106.099,E2 28106.099} C_VEL
LIN {X 0,Y 585.342,Z 289.298,A -85,B 0,C 180,E1 28102.709,E2 28102.709} C_VEL
LIN {X 0,Y 585.317,Z 324.735,A -85,B 0,C 180,E1 28099.978,E2 28099.978} C_VEL
LIN {X 0,Y 584.979,Z 366.942,A -85,B 0,C 180,E1 28096.688,E2 28096.688} C_VEL
LIN {X 0,Y 584.676,Z 409.349,A -85,B 0,C 180,E1 28093.449,E2 28093.449} C_VEL
LIN {X 0,Y 584.57,Z 436.481,A -85,B 0,C 180,E1 28091.433,E2 28091.433} C_VEL
LIN {X 0,Y 584.809,Z 462.775,A -85,B 0,C 180,E1 28091.097,E2 28091.097} C_VEL
LIN {X 0,Y 584.635,Z 578.886,A -85,B 0,C 180,E1 28089.625,E2 28089.625} C_VEL
LIN {X 0,Y 584.567,Z 596.076,A -85,B 0,C 180,E1 28089.203,E2 28089.203} C_VEL
LIN {X 0,Y 584.468,Z 610.889,A -85,B 0,C 180,E1 28088.659,E2 28088.659} C_VEL
LIN {X 0,Y 584.369,Z 625.911,A -85,B 0,C 180,E1 28087.917,E2 28087.917} C_VEL
LIN {X 0,Y 584.261,Z 639.766,A -85,B 0,C 180,E1 28087.029,E2 28087.029} C_VEL
LIN {X 0,Y 584.161,Z 652.671,A -85,B 0,C 180,E1 28085.993,E2 28085.993} C_VEL
LIN {X 0,Y 584.076,Z 664.446,A -85,B 0,C 180,E1 28084.812,E2 28084.812} C_VEL
LIN {X 0,Y 584.005,Z 674.687,A -85,B 0,C 180,E1 28083.534,E2 28083.534} C_VEL
LIN {X 0,Y 583.962,Z 684.015,A -85,B 0,C 180,E1 28082.061,E2 28082.061} C_VEL
LIN {X 0,Y 583.934,Z 691.118,A -85,B 0,C 180,E1 28080.589,E2 28080.589} C_VEL
LIN {X 0,Y 583.921,Z 696.686,A -85,B 0,C 180,E1 28079.019,E2 28079.019} C_VEL
LIN {X 0,Y 583.917,Z 700.301,A -85,B 0,C 180,E1 28077.449,E2 28077.449} C_VEL
LIN {X 0,Y 583.916,Z 702.178,A -85,B 0,C 180,E1 28075.876,E2 28075.876} C_VEL
LIN {X 0,Y 583.915,Z 702.271,A -85,B 0,C 180,E1 28074.197,E2 28074.197} C_VEL
LIN {X 0,Y 583.913,Z 700.567,A -85,B 0,C 180,E1 28072.622,E2 28072.622} C_VEL
LIN {X 0,Y 583.919,Z 697.11,A -85,B 0,C 180,E1 28071.036,E2 28071.036} C_VEL
LIN {X 0,Y 583.93,Z 692.009,A -85,B 0,C 180,E1 28069.543,E2 28069.543} C_VEL
LIN {X 0,Y 583.952,Z 685.577,A -85,B 0,C 180,E1 28068.143,E2 28068.143} C_VEL
LIN {X 0,Y 583.997,Z 677.226,A -85,B 0,C 180,E1 28066.737,E2 28066.737} C_VEL
LIN {X 0,Y 584.051,Z 667.261,A -85,B 0,C 180,E1 28065.425,E2 28065.425} C_VEL
LIN {X 0,Y 584.141,Z 655.842,A -85,B 0,C 180,E1 28064.208,E2 28064.208} C_VEL
LIN {X 0,Y 584.232,Z 643.219,A -85,B 0,C 180,E1 28063.137,E2 28063.137} C_VEL
LIN {X 0,Y 584.317,Z 630.52,A -85,B 0,C 180,E1 28062.267,E2 28062.267} C_VEL
LIN {X 0,Y 584.439,Z 616.421,A -85,B 0,C 180,E1 28061.497,E2 28061.497} C_VEL
LIN {X 0,Y 584.543,Z 600.56,A -85,B 0,C 180,E1 28060.854,E2 28060.854} C_VEL
LIN {X 0,Y 584.616,Z 584.142,A -85,B 0,C 180,E1 28060.392,E2 28060.392} C_VEL
LIN {X 0,Y 584.673,Z 566.093,A -85,B 0,C 180,E1 28060.099,E2 28060.099} C_VEL
LIN {X 0,Y 584.622,Z 436.777,A -85,B 0,C 180,E1 28058.482,E2 28058.482} C_VEL
LIN {X 0,Y 584.536,Z 435.4,A -85,B 0,C 180,E1 28058.423,E2 28058.423} C_VEL
LIN {X 0,Y 584.804,Z 391.798,A -85,B 0,C 180,E1 28055.128,E2 28055.128} C_VEL
LIN {X 0,Y 585.115,Z 348.616,A -85,B 0,C 180,E1 28051.802,E2 28051.802} C_VEL
LIN {X 0,Y 585.302,Z 313.981,A -85,B 0,C 180,E1 28049.114,E2 28049.114} C_VEL
LIN {X 0,Y 584.79,Z 274.585,A -85,B 0,C 180,E1 28046.295,E2 28046.295} C_VEL
LIN {X 0,Y 584.079,Z 239.981,A -85,B 0,C 180,E1 28044.003,E2 28044.003} C_VEL
LIN {X 0,Y 584.103,Z 239.999,A -85,B 0,C 180,E1 28040.98,E2 28040.98} C_VEL
LIN {X 0,Y 585.226,Z 243.186,A -85,B 0,C 180,E1 28040.665,E2 28040.665} C_VEL
LIN {X 0,Y 588.337,Z 249.616,A -85,B 0,C 180,E1 28039.966,E2 28039.966} C_VEL
LIN {X 0,Y 588.123,Z 307.411,A -85,B 0,C 180,E1 28036.265,E2 28036.265} C_VEL
LIN {X 0,Y 589.797,Z 318.936,A -85,B 0,C 180,E1 28035.426,E2 28035.426} C_VEL
LIN {X 0,Y 592.528,Z 327.096,A -85,B 0,C 180,E1 28034.732,E2 28034.732} C_VEL
LIN {X 0,Y 595.268,Z 331.671,A -85,B 0,C 180,E1 28034.193,E2 28034.193} C_VEL
LIN {X 0,Y 597.406,Z 334.013,A -85,B 0,C 180,E1 28033.696,E2 28033.696} C_VEL
LIN {X 0,Y 599.119,Z 334.943,A -85,B 0,C 180,E1 28033.173,E2 28033.173} C_VEL
LIN {X 0,Y 600.251,Z 334.354,A -85,B 0,C 180,E1 28032.587,E2 28032.587} C_VEL
LIN {X 0,Y 600.379,Z 332.197,A -85,B 0,C 180,E1 28032.033,E2 28032.033} C_VEL
LIN {X 0,Y 599.505,Z 328.697,A -85,B 0,C 180,E1 28031.558,E2 28031.558} C_VEL
LIN {X 0,Y 597.719,Z 323.952,A -85,B 0,C 180,E1 28031.178,E2 28031.178} C_VEL
LIN {X 0,Y 594.958,Z 316.372,A -85,B 0,C 180,E1 28030.856,E2 28030.856} C_VEL
LIN {X 0,Y 593.041,Z 306.958,A -85,B 0,C 180,E1 28030.641,E2 28030.641} C_VEL
LIN {X 0,Y 592.101,Z 294.902,A -85,B 0,C 180,E1 28030.535,E2 28030.535} C_VEL
LIN {X 0,Y 591.862,Z 250.734,A -85,B 0,C 180,E1 28030.508,E2 28030.508} C_VEL
LIN {X 0,Y 588.95,Z 246.911,A -85,B 0,C 180,E1 28030.175,E2 28030.175} C_VEL
LIN {X 0,Y 588.306,Z 246.069,A -85,B 0,C 180,E1 28030.101,E2 28030.101} C_VEL
LIN {X 0,Y 585.497,Z 243.639,A -85,B 0,C 180,E1 28029.774,E2 28029.774} C_VEL
LIN {X 0,Y 584.18,Z 240.676,A -85,B 0,C 180,E1 28029.618,E2 28029.618} C_VEL
LIN {X 0,Y 584.061,Z 239.984,A -85,B 0,C 180,E1 28029.588,E2 28029.588} C_VEL
LIN {X 0,Y 584.076,Z 240.099,A -85,B 0,C 180,E1 28027.732,E2 28027.732} C_VEL
LIN {X 0,Y 585.39,Z 243.476,A -85,B 0,C 180,E1 28027.418,E2 28027.418} C_VEL
LIN {X 0,Y 587.521,Z 248.792,A -85,B 0,C 180,E1 28026.924,E2 28026.924} C_VEL
LIN {X 0,Y 586.973,Z 299.152,A -85,B 0,C 180,E1 28023.85,E2 28023.85} C_VEL
LIN {X 0,Y 587.101,Z 302.901,A -85,B 0,C 180,E1 28023.657,E2 28023.657} C_VEL
LIN {X 0,Y 587.705,Z 308.067,A -85,B 0,C 180,E1 28023.543,E2 28023.543} C_VEL
LIN {X 0,Y 587.047,Z 528.23,A -85,B 0,C 180,E1 28020.473,E2 28020.473} C_VEL
LIN {X 0,Y 586.805,Z 608.956,A -85,B 0,C 180,E1 28019.339,E2 28019.339} C_VEL
LIN {X 0,Y 586.619,Z 630.704,A -85,B 0,C 180,E1 28018.843,E2 28018.843} C_VEL
LIN {X 0,Y 586.355,Z 653.12,A -85,B 0,C 180,E1 28018.137,E2 28018.137} C_VEL
LIN {X 0,Y 586.123,Z 674.1,A -85,B 0,C 180,E1 28017.282,E2 28017.282} C_VEL
LIN {X 0,Y 585.824,Z 693.747,A -85,B 0,C 180,E1 28016.289,E2 28016.289} C_VEL
LIN {X 0,Y 585.486,Z 714.145,A -85,B 0,C 180,E1 28015.057,E2 28015.057} C_VEL
LIN {X 0,Y 585.205,Z 733.359,A -85,B 0,C 180,E1 28013.682,E2 28013.682} C_VEL
LIN {X 0,Y 584.927,Z 751.102,A -85,B 0,C 180,E1 28012.196,E2 28012.196} C_VEL
LIN {X 0,Y 584.661,Z 768.222,A -85,B 0,C 180,E1 28010.523,E2 28010.523} C_VEL
LIN {X 0,Y 584.437,Z 783.724,A -85,B 0,C 180,E1 28008.762,E2 28008.762} C_VEL
LIN {X 0,Y 584.255,Z 797.751,A -85,B 0,C 180,E1 28006.914,E2 28006.914} C_VEL
LIN {X 0,Y 584.131,Z 810.344,A -85,B 0,C 180,E1 28004.979,E2 28004.979} C_VEL
LIN {X 0,Y 584.036,Z 820.855,A -85,B 0,C 180,E1 28003.061,E2 28003.061} C_VEL
LIN {X 0,Y 583.966,Z 830.483,A -85,B 0,C 180,E1 28000.956,E2 28000.956} C_VEL
LIN {X 0,Y 583.94,Z 838.157,A -85,B 0,C 180,E1 27998.896,E2 27998.896} C_VEL
LIN {X 0,Y 583.926,Z 844.171,A -85,B 0,C 180,E1 27996.785,E2 27996.785} C_VEL
LIN {X 0,Y 583.916,Z 848.629,A -85,B 0,C 180,E1 27994.616,E2 27994.616} C_VEL
LIN {X 0,Y 583.908,Z 851.418,A -85,B 0,C 180,E1 27992.453,E2 27992.453} C_VEL
LIN {X 0,Y 583.9,Z 852.448,A -85,B 0,C 180,E1 27990.294,E2 27990.294} C_VEL
LIN {X 0,Y 583.906,Z 851.82,A -85,B 0,C 180,E1 27988.136,E2 27988.136} C_VEL
LIN {X 0,Y 583.912,Z 849.58,A -85,B 0,C 180,E1 27985.974,E2 27985.974} C_VEL
LIN {X 0,Y 583.918,Z 845.788,A -85,B 0,C 180,E1 27983.906,E2 27983.906} C_VEL
LIN {X 0,Y 583.935,Z 840.185,A -85,B 0,C 180,E1 27981.766,E2 27981.766} C_VEL
LIN {X 0,Y 583.967,Z 833.318,A -85,B 0,C 180,E1 27979.743,E2 27979.743} C_VEL
LIN {X 0,Y 584.01,Z 824.758,A -85,B 0,C 180,E1 27977.743,E2 27977.743} C_VEL
LIN {X 0,Y 584.1,Z 813.825,A -85,B 0,C 180,E1 27975.628,E2 27975.628} C_VEL
LIN {X 0,Y 584.226,Z 801.993,A -85,B 0,C 180,E1 27973.699,E2 27973.699} C_VEL
LIN {X 0,Y 584.377,Z 788.689,A -85,B 0,C 180,E1 27971.856,E2 27971.856} C_VEL
LIN {X 0,Y 584.561,Z 773.962,A -85,B 0,C 180,E1 27970.1,E2 27970.1} C_VEL
LIN {X 0,Y 584.81,Z 757.252,A -85,B 0,C 180,E1 27968.38,E2 27968.38} C_VEL
LIN {X 0,Y 585.104,Z 739.8,A -85,B 0,C 180,E1 27966.833,E2 27966.833} C_VEL
LIN {X 0,Y 585.408,Z 721.287,A -85,B 0,C 180,E1 27965.424,E2 27965.424} C_VEL
LIN {X 0,Y 585.679,Z 702.198,A -85,B 0,C 180,E1 27964.193,E2 27964.193} C_VEL
LIN {X 0,Y 585.987,Z 681.284,A -85,B 0,C 180,E1 27963.062,E2 27963.062} C_VEL
LIN {X 0,Y 586.3,Z 660.547,A -85,B 0,C 180,E1 27962.142,E2 27962.142} C_VEL
LIN {X 0,Y 586.522,Z 639.125,A -85,B 0,C 180,E1 27961.397,E2 27961.397} C_VEL
LIN {X 0,Y 586.733,Z 617.306,A -85,B 0,C 180,E1 27960.831,E2 27960.831} C_VEL
LIN {X 0,Y 586.876,Z 595.172,A -85,B 0,C 180,E1 27960.444,E2 27960.444} C_VEL
LIN {X 0,Y 587.482,Z 369.833,A -85,B 0,C 180,E1 27957.326,E2 27957.326} C_VEL
LIN {X 0,Y 587.501,Z 306.656,A -85,B 0,C 180,E1 27956.423,E2 27956.423} C_VEL
LIN {X 0,Y 586.704,Z 302.65,A -85,B 0,C 180,E1 27956.303,E2 27956.303} C_VEL
LIN {X 0,Y 587.174,Z 260.921,A -85,B 0,C 180,E1 27953.324,E2 27953.324} C_VEL
LIN {X 0,Y 587.16,Z 247.855,A -85,B 0,C 180,E1 27952.357,E2 27952.357} C_VEL
LIN {X 0,Y 584.093,Z 239.98,A -85,B 0,C 180,E1 27951.519,E2 27951.519} C_VEL
LIN {X 0,Y 584.101,Z 240.215,A -85,B 0,C 180,E1 27950.391,E2 27950.391} C_VEL
LIN {X 0,Y 585.258,Z 243.295,A -85,B 0,C 180,E1 27950.255,E2 27950.255} C_VEL
LIN {X 0,Y 587.662,Z 245.712,A -85,B 0,C 180,E1 27949.974,E2 27949.974} C_VEL
LIN {X 0,Y 588.869,Z 246.762,A -85,B 0,C 180,E1 27949.834,E2 27949.834} C_VEL
LIN {X 0,Y 591.7,Z 250.589,A -85,B 0,C 180,E1 27949.51,E2 27949.51} C_VEL
LIN {X 0,Y 592.028,Z 250.894,A -85,B 0,C 180,E1 27949.473,E2 27949.473} C_VEL
LIN {X 0,Y 592.209,Z 336.105,A -85,B 0,C 180,E1 27949.453,E2 27949.453} C_VEL
LIN {X 0,Y 593.348,Z 346.95,A -85,B 0,C 180,E1 27949.324,E2 27949.324} C_VEL
LIN {X 0,Y 595.45,Z 355.607,A -85,B 0,C 180,E1 27949.089,E2 27949.089} C_VEL
LIN {X 0,Y 597.713,Z 361.833,A -85,B 0,C 180,E1 27948.785,E2 27948.785} C_VEL
LIN {X 0,Y 599.095,Z 366.376,A -85,B 0,C 180,E1 27948.375,E2 27948.375} C_VEL
LIN {X 0,Y 599.53,Z 369.497,A -85,B 0,C 180,E1 27947.899,E2 27947.899} C_VEL
LIN {X 0,Y 599.037,Z 371.349,A -85,B 0,C 180,E1 27947.339,E2 27947.339} C_VEL
LIN {X 0,Y 597.827,Z 371.706,A -85,B 0,C 180,E1 27946.819,E2 27946.819} C_VEL
LIN {X 0,Y 595.944,Z 370.608,A -85,B 0,C 180,E1 27946.271,E2 27946.271} C_VEL
LIN {X 0,Y 593.559,Z 367.763,A -85,B 0,C 180,E1 27945.718,E2 27945.718} C_VEL
LIN {X 0,Y 590.892,Z 362.7,A -85,B 0,C 180,E1 27945.153,E2 27945.153} C_VEL
LIN {X 0,Y 588.307,Z 353.092,A -85,B 0,C 180,E1 27944.308,E2 27944.308} C_VEL
LIN {X 0,Y 587.231,Z 340.806,A -85,B 0,C 180,E1 27943.361,E2 27943.361} C_VEL
LIN {X 0,Y 587.719,Z 292.934,A -85,B 0,C 180,E1 27939.89,E2 27939.89} C_VEL
LIN {X 0,Y 588.238,Z 256.769,A -85,B 0,C 180,E1 27937.137,E2 27937.137} C_VEL
LIN {X 0,Y 588.401,Z 250.077,A -85,B 0,C 180,E1 27936.616,E2 27936.616} C_VEL
LIN {X 0,Y 585.216,Z 243.192,A -85,B 0,C 180,E1 27935.751,E2 27935.751} C_VEL
LIN {X 0,Y 584.098,Z 239.982,A -85,B 0,C 180,E1 27935.351,E2 27935.351} C_VEL
LIN {X 0,Y 584.097,Z 239.982,A -85,B 0,C 180,E1 27932.05,E2 27932.05} C_VEL
LIN {X 0,Y 584.096,Z 239.978,A -85,B 0,C 180,E1 27928.752,E2 27928.752} C_VEL
LIN {X 0,Y 584.09,Z 239.991,A -85,B 0,C 180,E1 27926.477,E2 27926.477} C_VEL
LIN {X 0,Y 584.458,Z 254.006,A -85,B 0,C 180,E1 27925.597,E2 27925.597} C_VEL
LIN {X 0,Y 584.955,Z 296.59,A -85,B 0,C 180,E1 27922.83,E2 27922.83} C_VEL
LIN {X 0,Y 585.204,Z 335.976,A -85,B 0,C 180,E1 27920.137,E2 27920.137} C_VEL
LIN {X 0,Y 584.985,Z 377.445,A -85,B 0,C 180,E1 27917.166,E2 27917.166} C_VEL
LIN {X 0,Y 584.672,Z 424.189,A -85,B 0,C 180,E1 27913.852,E2 27913.852} C_VEL
LIN {X 0,Y 584.419,Z 472.31,A -85,B 0,C 180,E1 27910.498,E2 27910.498} C_VEL
LIN {X 0,Y 584.395,Z 486.06,A -85,B 0,C 180,E1 27909.574,E2 27909.574} C_VEL
LIN {X 0,Y 584.422,Z 600.114,A -85,B 0,C 180,E1 27908.139,E2 27908.139} C_VEL
LIN {X 0,Y 584.348,Z 614.839,A -85,B 0,C 180,E1 27907.768,E2 27907.768} C_VEL
LIN {X 0,Y 584.277,Z 630.069,A -85,B 0,C 180,E1 27907.176,E2 27907.176} C_VEL
LIN {X 0,Y 584.182,Z 642.917,A -85,B 0,C 180,E1 27906.486,E2 27906.486} C_VEL
LIN {X 0,Y 584.122,Z 655.544,A -85,B 0,C 180,E1 27905.599,E2 27905.599} C_VEL
LIN {X 0,Y 584.052,Z 666.483,A -85,B 0,C 180,E1 27904.615,E2 27904.615} C_VEL
LIN {X 0,Y 583.994,Z 676.836,A -85,B 0,C 180,E1 27903.435,E2 27903.435} C_VEL
LIN {X 0,Y 583.955,Z 684.856,A -85,B 0,C 180,E1 27902.257,E2 27902.257} C_VEL
LIN {X 0,Y 583.931,Z 692.039,A -85,B 0,C 180,E1 27900.883,E2 27900.883} C_VEL
LIN {X 0,Y 583.923,Z 697.118,A -85,B 0,C 180,E1 27899.509,E2 27899.509} C_VEL
LIN {X 0,Y 583.918,Z 700.511,A -85,B 0,C 180,E1 27898.135,E2 27898.135} C_VEL
LIN {X 0,Y 583.917,Z 702.277,A -85,B 0,C 180,E1 27896.657,E2 27896.657} C_VEL
LIN {X 0,Y 583.917,Z 702.234,A -85,B 0,C 180,E1 27895.187,E2 27895.187} C_VEL
LIN {X 0,Y 583.917,Z 700.372,A -85,B 0,C 180,E1 27893.708,E2 27893.708} C_VEL
LIN {X 0,Y 583.922,Z 696.882,A -85,B 0,C 180,E1 27892.324,E2 27892.324} C_VEL
LIN {X 0,Y 583.933,Z 691.617,A -85,B 0,C 180,E1 27890.936,E2 27890.936} C_VEL
LIN {X 0,Y 583.955,Z 684.791,A -85,B 0,C 180,E1 27889.642,E2 27889.642} C_VEL
LIN {X 0,Y 583.995,Z 676.595,A -85,B 0,C 180,E1 27888.444,E2 27888.444} C_VEL
LIN {X 0,Y 584.04,Z 668.656,A -85,B 0,C 180,E1 27887.516,E2 27887.516} C_VEL
LIN {X 0,Y 583.09,Z 663.365,A -85,B 0,C 180,E1 27886.964,E2 27886.964} C_VEL
LIN {X 0,Y 579.081,Z 654.079,A -85,B 0,C 180,E1 27886.09,E2 27886.09} C_VEL
LIN {X 0,Y 576.786,Z 647.286,A -85,B 0,C 180,E1 27885.562,E2 27885.562} C_VEL
LIN {X 0,Y 576.288,Z 642.657,A -85,B 0,C 180,E1 27885.262,E2 27885.262} C_VEL
LIN {X 0,Y 576.399,Z 630.648,A -85,B 0,C 180,E1 27884.609,E2 27884.609} C_VEL
LIN {X 0,Y 576.496,Z 616.358,A -85,B 0,C 180,E1 27884.026,E2 27884.026} C_VEL
LIN {X 0,Y 576.597,Z 601.299,A -85,B 0,C 180,E1 27883.626,E2 27883.626} C_VEL
LIN {X 0,Y 576.643,Z 569.007,A -85,B 0,C 180,E1 27883.189,E2 27883.189} C_VEL
LIN {X 0,Y 576.524,Z 485.8,A -85,B 0,C 180,E1 27882.143,E2 27882.143} C_VEL
LIN {X 0,Y 576.817,Z 439.799,A -85,B 0,C 180,E1 27878.919,E2 27878.919} C_VEL
LIN {X 0,Y 577.211,Z 394.061,A -85,B 0,C 180,E1 27875.652,E2 27875.652} C_VEL
LIN {X 0,Y 577.568,Z 348.392,A -85,B 0,C 180,E1 27872.357,E2 27872.357} C_VEL
LIN {X 0,Y 577.641,Z 315.916,A -85,B 0,C 180,E1 27870.041,E2 27870.041} C_VEL
LIN {X 0,Y 577.635,Z 270.454,A -85,B 0,C 180,E1 27866.78,E2 27866.78} C_VEL
LIN {X 0,Y 577.545,Z 246.097,A -85,B 0,C 180,E1 27865.059,E2 27865.059} C_VEL
LIN {X 0,Y 576.131,Z 240.973,A -85,B 0,C 180,E1 27864.607,E2 27864.607} C_VEL
LIN {X 0,Y 576.15,Z 240.972,A -85,B 0,C 180,E1 27861.347,E2 27861.347} C_VEL
LIN {X 0,Y 576.151,Z 240.968,A -85,B 0,C 180,E1 27858.076,E2 27858.076} C_VEL
LIN {X 0,Y 576.134,Z 240.972,A -85,B 0,C 180,E1 27854.639,E2 27854.639} C_VEL
LIN {X 0,Y 576.151,Z 240.971,A -85,B 0,C 180,E1 27851.391,E2 27851.391} C_VEL
LIN {X 0,Y 576.142,Z 240.97,A -85,B 0,C 180,E1 27848.157,E2 27848.157} C_VEL
LIN {X 0,Y 576.175,Z 241.078,A -85,B 0,C 180,E1 27847.571,E2 27847.571} C_VEL
LIN {X 0,Y 579.092,Z 249.998,A -85,B 0,C 180,E1 27846.561,E2 27846.561} C_VEL
LIN {X 0,Y 578.53,Z 285.859,A -85,B 0,C 180,E1 27843.409,E2 27843.409} C_VEL
LIN {X 0,Y 578.442,Z 300.705,A -85,B 0,C 180,E1 27842.156,E2 27842.156} C_VEL
LIN {X 0,Y 579.631,Z 307.35,A -85,B 0,C 180,E1 27841.998,E2 27841.998} C_VEL
LIN {X 0,Y 578.928,Z 538.317,A -85,B 0,C 180,E1 27838.872,E2 27838.872} C_VEL
LIN {X 0,Y 578.775,Z 565.522,A -85,B 0,C 180,E1 27838.452,E2 27838.452} C_VEL
LIN {X 0,Y 578.569,Z 585.606,A -85,B 0,C 180,E1 27837.96,E2 27837.96} C_VEL
LIN {X 0,Y 578.32,Z 605.21,A -85,B 0,C 180,E1 27837.294,E2 27837.294} C_VEL
LIN {X 0,Y 578.026,Z 624.555,A -85,B 0,C 180,E1 27836.45,E2 27836.45} C_VEL
LIN {X 0,Y 577.682,Z 643.518,A -85,B 0,C 180,E1 27835.42,E2 27835.42} C_VEL
LIN {X 0,Y 577.362,Z 661.651,A -85,B 0,C 180,E1 27834.232,E2 27834.232} C_VEL
LIN {X 0,Y 577.046,Z 678.737,A -85,B 0,C 180,E1 27832.892,E2 27832.892} C_VEL
LIN {X 0,Y 576.774,Z 694.391,A -85,B 0,C 180,E1 27831.456,E2 27831.456} C_VEL
LIN {X 0,Y 576.505,Z 709.88,A -85,B 0,C 180,E1 27829.767,E2 27829.767} C_VEL
LIN {X 0,Y 576.307,Z 723.249,A -85,B 0,C 180,E1 27828.055,E2 27828.055} C_VEL
LIN {X 0,Y 576.157,Z 735.252,A -85,B 0,C 180,E1 27826.224,E2 27826.224} C_VEL
LIN {X 0,Y 576.046,Z 745.158,A -85,B 0,C 180,E1 27824.409,E2 27824.409} C_VEL
LIN {X 0,Y 575.977,Z 754.049,A -85,B 0,C 180,E1 27822.431,E2 27822.431} C_VEL
LIN {X 0,Y 575.938,Z 761.208,A -85,B 0,C 180,E1 27820.402,E2 27820.402} C_VEL
LIN {X 0,Y 575.92,Z 766.543,A -85,B 0,C 180,E1 27818.386,E2 27818.386} C_VEL
LIN {X 0,Y 575.91,Z 770.133,A -85,B 0,C 180,E1 27816.38,E2 27816.38} C_VEL
LIN {X 0,Y 575.907,Z 772.053,A -85,B 0,C 180,E1 27814.381,E2 27814.381} C_VEL
LIN {X 0,Y 575.904,Z 772.368,A -85,B 0,C 180,E1 27812.289,E2 27812.289} C_VEL
LIN {X 0,Y 575.911,Z 770.933,A -85,B 0,C 180,E1 27810.199,E2 27810.199} C_VEL
LIN {X 0,Y 575.919,Z 767.743,A -85,B 0,C 180,E1 27808.11,E2 27808.11} C_VEL
LIN {X 0,Y 575.935,Z 763.029,A -85,B 0,C 180,E1 27806.118,E2 27806.118} C_VEL
LIN {X 0,Y 575.966,Z 756.506,A -85,B 0,C 180,E1 27804.109,E2 27804.109} C_VEL
LIN {X 0,Y 576.009,Z 748.609,A -85,B 0,C 180,E1 27802.218,E2 27802.218} C_VEL
LIN {X 0,Y 576.098,Z 738.841,A -85,B 0,C 180,E1 27800.308,E2 27800.308} C_VEL
LIN {X 0,Y 576.239,Z 727.604,A -85,B 0,C 180,E1 27798.49,E2 27798.49} C_VEL
LIN {X 0,Y 576.43,Z 715.012,A -85,B 0,C 180,E1 27796.764,E2 27796.764} C_VEL
LIN {X 0,Y 576.668,Z 699.932,A -85,B 0,C 180,E1 27795.028,E2 27795.028} C_VEL
LIN {X 0,Y 576.945,Z 684.74,A -85,B 0,C 180,E1 27793.54,E2 27793.54} C_VEL
LIN {X 0,Y 577.269,Z 667.309,A -85,B 0,C 180,E1 27792.095,E2 27792.095} C_VEL
LIN {X 0,Y 577.577,Z 650.18,A -85,B 0,C 180,E1 27790.902,E2 27790.902} C_VEL
LIN {X 0,Y 577.897,Z 631.429,A -85,B 0,C 180,E1 27789.808,E2 27789.808} C_VEL
LIN {X 0,Y 578.197,Z 612.65,A -85,B 0,C 180,E1 27788.919,E2 27788.919} C_VEL
LIN {X 0,Y 578.499,Z 592.478,A -85,B 0,C 180,E1 27788.162,E2 27788.162} C_VEL
LIN {X 0,Y 578.714,Z 572.28,A -85,B 0,C 180,E1 27787.603,E2 27787.603} C_VEL
LIN {X 0,Y 578.863,Z 552.303,A -85,B 0,C 180,E1 27787.229,E2 27787.229} C_VEL
LIN {X 0,Y 579.647,Z 312.109,A -85,B 0,C 180,E1 27783.979,E2 27783.979} C_VEL
LIN {X 0,Y 579.45,Z 303.553,A -85,B 0,C 180,E1 27783.849,E2 27783.849} C_VEL
LIN {X 0,Y 578.626,Z 298.918,A -85,B 0,C 180,E1 27783.717,E2 27783.717} C_VEL
LIN {X 0,Y 579.24,Z 253.704,A -85,B 0,C 180,E1 27780.36,E2 27780.36} C_VEL
LIN {X 0,Y 579.257,Z 249.715,A -85,B 0,C 180,E1 27780.056,E2 27780.056} C_VEL
LIN {X 0,Y 576.143,Z 240.972,A -85,B 0,C 180,E1 27779.154,E2 27779.154} C_VEL
LIN {X 0,Y 576.135,Z 240.971,A -85,B 0,C 180,E1 27775.876,E2 27775.876} C_VEL
LIN {X 0,Y 576.159,Z 240.971,A -85,B 0,C 180,E1 27772.638,E2 27772.638} C_VEL
LIN {X 0,Y 576.156,Z 240.972,A -85,B 0,C 180,E1 27769.269,E2 27769.269} C_VEL
LIN {X 0,Y 576.159,Z 240.97,A -85,B 0,C 180,E1 27765.763,E2 27765.763} C_VEL
LIN {X 0,Y 576.144,Z 240.971,A -85,B 0,C 180,E1 27762.461,E2 27762.461} C_VEL
LIN {X 0,Y 576.133,Z 240.97,A -85,B 0,C 180,E1 27759.283,E2 27759.283} C_VEL
LIN {X 0,Y 576.157,Z 240.968,A -85,B 0,C 180,E1 27756.031,E2 27756.031} C_VEL
LIN {X 0,Y 576.159,Z 240.971,A -85,B 0,C 180,E1 27752.664,E2 27752.664} C_VEL
LIN {X 0,Y 576.159,Z 240.971,A -85,B 0,C 180,E1 27749.186,E2 27749.186} C_VEL
LIN {X 0,Y 576.162,Z 241.044,A -85,B 0,C 180,E1 27746.835,E2 27746.835} C_VEL
LIN {X 0,Y 577.747,Z 247.064,A -85,B 0,C 180,E1 27746.298,E2 27746.298} C_VEL
LIN {X 0,Y 577.787,Z 293.667,A -85,B 0,C 180,E1 27742.7,E2 27742.7} C_VEL
LIN {X 0,Y 577.667,Z 332.038,A -85,B 0,C 180,E1 27739.726,E2 27739.726} C_VEL
LIN {X 0,Y 577.31,Z 372.523,A -85,B 0,C 180,E1 27736.553,E2 27736.553} C_VEL
LIN {X 0,Y 576.908,Z 415.617,A -85,B 0,C 180,E1 27733.225,E2 27733.225} C_VEL
LIN {X 0,Y 576.789,Z 436.427,A -85,B 0,C 180,E1 27731.663,E2 27731.663} C_VEL
LIN {X 0,Y 577.147,Z 444.513,A -85,B 0,C 180,E1 27731.549,E2 27731.549} C_VEL
LIN {X 0,Y 576.89,Z 578.499,A -85,B 0,C 180,E1 27729.832,E2 27729.832} C_VEL
LIN {X 0,Y 576.8,Z 595.907,A -85,B 0,C 180,E1 27729.403,E2 27729.403} C_VEL
LIN {X 0,Y 576.676,Z 610.158,A -85,B 0,C 180,E1 27728.877,E2 27728.877} C_VEL
LIN {X 0,Y 576.552,Z 624.526,A -85,B 0,C 180,E1 27728.176,E2 27728.176} C_VEL
LIN {X 0,Y 576.388,Z 638.666,A -85,B 0,C 180,E1 27727.275,E2 27727.275} C_VEL
LIN {X 0,Y 576.267,Z 651.212,A -85,B 0,C 180,E1 27726.276,E2 27726.276} C_VEL
LIN {X 0,Y 576.135,Z 664.187,A -85,B 0,C 180,E1 27724.978,E2 27724.978} C_VEL
LIN {X 0,Y 576.049,Z 673.747,A -85,B 0,C 180,E1 27723.782,E2 27723.782} C_VEL
LIN {X 0,Y 575.983,Z 682.738,A -85,B 0,C 180,E1 27722.388,E2 27722.388} C_VEL
LIN {X 0,Y 575.941,Z 690.148,A -85,B 0,C 180,E1 27720.896,E2 27720.896} C_VEL
LIN {X 0,Y 575.925,Z 695.697,A -85,B 0,C 180,E1 27719.404,E2 27719.404} C_VEL
LIN {X 0,Y 575.917,Z 699.913,A -85,B 0,C 180,E1 27717.712,E2 27717.712} C_VEL
LIN {X 0,Y 575.916,Z 702.007,A -85,B 0,C 180,E1 27716.118,E2 27716.118} C_VEL
LIN {X 0,Y 575.916,Z 702.398,A -85,B 0,C 180,E1 27714.421,E2 27714.421} C_VEL
LIN {X 0,Y 575.917,Z 700.912,A -85,B 0,C 180,E1 27712.82,E2 27712.82} C_VEL
LIN {X 0,Y 575.919,Z 697.956,A -85,B 0,C 180,E1 27711.313,E2 27711.313} C_VEL
LIN {X 0,Y 575.935,Z 692.939,A -85,B 0,C 180,E1 27709.7,E2 27709.7} C_VEL
LIN {X 0,Y 575.96,Z 686.668,A -85,B 0,C 180,E1 27708.266,E2 27708.266} C_VEL
LIN {X 0,Y 576.011,Z 678.727,A -85,B 0,C 180,E1 27706.857,E2 27706.857} C_VEL
LIN {X 0,Y 576.087,Z 669.2,A -85,B 0,C 180,E1 27705.527,E2 27705.527} C_VEL
LIN {X 0,Y 576.181,Z 659.112,A -85,B 0,C 180,E1 27704.389,E2 27704.389} C_VEL
LIN {X 0,Y 576.325,Z 646.276,A -85,B 0,C 180,E1 27703.211,E2 27703.211} C_VEL
LIN {X 0,Y 576.438,Z 633.423,A -85,B 0,C 180,E1 27702.277,E2 27702.277} C_VEL
LIN {X 0,Y 576.583,Z 620.073,A -85,B 0,C 180,E1 27701.498,E2 27701.498} C_VEL
LIN {X 0,Y 576.741,Z 604.346,A -85,B 0,C 180,E1 27700.795,E2 27700.795} C_VEL
LIN {X 0,Y 576.852,Z 588.217,A -85,B 0,C 180,E1 27700.287,E2 27700.287} C_VEL
LIN {X 0,Y 576.925,Z 571.651,A -85,B 0,C 180,E1 27699.968,E2 27699.968} C_VEL
LIN {X 0,Y 576.943,Z 437.506,A -85,B 0,C 180,E1 27698.266,E2 27698.266} C_VEL
LIN {X 0,Y 576.756,Z 435.802,A -85,B 0,C 180,E1 27698.224,E2 27698.224} C_VEL
LIN {X 0,Y 577.124,Z 392.195,A -85,B 0,C 180,E1 27694.884,E2 27694.884} C_VEL
LIN {X 0,Y 577.525,Z 349.122,A -85,B 0,C 180,E1 27691.525,E2 27691.525} C_VEL
LIN {X 0,Y 577.547,Z 314.285,A -85,B 0,C 180,E1 27688.895,E2 27688.895} C_VEL
LIN {X 0,Y 577.019,Z 277.952,A -85,B 0,C 180,E1 27686.324,E2 27686.324} C_VEL
LIN {X 0,Y 576.393,Z 245.497,A -85,B 0,C 180,E1 27684.192,E2 27684.192} C_VEL
LIN {X 0,Y 576.141,Z 240.97,A -85,B 0,C 180,E1 27683.891,E2 27683.891} C_VEL
LIN {X 0,Y 576.167,Z 241.118,A -85,B 0,C 180,E1 27681.611,E2 27681.611} C_VEL
LIN {X 0,Y 577.291,Z 244.181,A -85,B 0,C 180,E1 27681.3,E2 27681.3} C_VEL
LIN {X 0,Y 581.871,Z 253.46,A -85,B 0,C 180,E1 27680.266,E2 27680.266} C_VEL
LIN {X 0,Y 581.408,Z 310.034,A -85,B 0,C 180,E1 27676.605,E2 27676.605} C_VEL
LIN {X 0,Y 583.021,Z 321.906,A -85,B 0,C 180,E1 27675.734,E2 27675.734} C_VEL
LIN {X 0,Y 585.606,Z 330.362,A -85,B 0,C 180,E1 27675.02,E2 27675.02} C_VEL
LIN {X 0,Y 589.108,Z 336.537,A -85,B 0,C 180,E1 27674.395,E2 27674.395} C_VEL
LIN {X 0,Y 592.332,Z 340.09,A -85,B 0,C 180,E1 27673.882,E2 27673.882} C_VEL
LIN {X 0,Y 595.068,Z 341.953,A -85,B 0,C 180,E1 27673.319,E2 27673.319} C_VEL
LIN {X 0,Y 597.07,Z 342.183,A -85,B 0,C 180,E1 27672.705,E2 27672.705} C_VEL
LIN {X 0,Y 597.955,Z 340.817,A -85,B 0,C 180,E1 27672.108,E2 27672.108} C_VEL
LIN {X 0,Y 597.65,Z 338.078,A -85,B 0,C 180,E1 27671.555,E2 27671.555} C_VEL
LIN {X 0,Y 596.16,Z 333.998,A -85,B 0,C 180,E1 27671.074,E2 27671.074} C_VEL
LIN {X 0,Y 593.571,Z 328.668,A -85,B 0,C 180,E1 27670.701,E2 27670.701} C_VEL
LIN {X 0,Y 590.444,Z 320.442,A -85,B 0,C 180,E1 27670.347,E2 27670.347} C_VEL
LIN {X 0,Y 588.286,Z 310.743,A -85,B 0,C 180,E1 27670.099,E2 27670.099} C_VEL
LIN {X 0,Y 587.074,Z 298.657,A -85,B 0,C 180,E1 27669.958,E2 27669.958} C_VEL
LIN {X 0,Y 586.857,Z 278.809,A -85,B 0,C 180,E1 27669.933,E2 27669.933} C_VEL
LIN {X 0,Y 586.698,Z 254.751,A -85,B 0,C 180,E1 27669.914,E2 27669.914} C_VEL
LIN {X 0,Y 584.938,Z 252.551,A -85,B 0,C 180,E1 27669.708,E2 27669.708} C_VEL
LIN {X 0,Y 581.756,Z 249.098,A -85,B 0,C 180,E1 27669.329,E2 27669.329} C_VEL
LIN {X 0,Y 580.649,Z 247.221,A -85,B 0,C 180,E1 27669.195,E2 27669.195} C_VEL
LIN {X 0,Y 577.816,Z 244.958,A -85,B 0,C 180,E1 27668.85,E2 27668.85} C_VEL
LIN {X 0,Y 576.329,Z 241.922,A -85,B 0,C 180,E1 27668.666,E2 27668.666} C_VEL
LIN {X 0,Y 576.15,Z 240.972,A -85,B 0,C 180,E1 27668.627,E2 27668.627} C_VEL
LIN {X 0,Y 576.138,Z 241.045,A -85,B 0,C 180,E1 27668.284,E2 27668.284} C_VEL
LIN {X 0,Y 577.254,Z 244.192,A -85,B 0,C 180,E1 27667.992,E2 27667.992} C_VEL
LIN {X 0,Y 580.756,Z 251.934,A -85,B 0,C 180,E1 27667.226,E2 27667.226} C_VEL
LIN {X 0,Y 580.053,Z 302.189,A -85,B 0,C 180,E1 27664.132,E2 27664.132} C_VEL
LIN {X 0,Y 581.029,Z 309.188,A -85,B 0,C 180,E1 27663.964,E2 27663.964} C_VEL
LIN {X 0,Y 580.146,Z 529.315,A -85,B 0,C 180,E1 27660.86,E2 27660.86} C_VEL
LIN {X 0,Y 579.823,Z 608.944,A -85,B 0,C 180,E1 27659.728,E2 27659.728} C_VEL
LIN {X 0,Y 579.571,Z 630.849,A -85,B 0,C 180,E1 27659.224,E2 27659.224} C_VEL
LIN {X 0,Y 579.234,Z 652.882,A -85,B 0,C 180,E1 27658.524,E2 27658.524} C_VEL
LIN {X 0,Y 578.912,Z 674.064,A -85,B 0,C 180,E1 27657.652,E2 27657.652} C_VEL
LIN {X 0,Y 578.501,Z 693.754,A -85,B 0,C 180,E1 27656.648,E2 27656.648} C_VEL
LIN {X 0,Y 578.066,Z 714.151,A -85,B 0,C 180,E1 27655.402,E2 27655.402} C_VEL
LIN {X 0,Y 577.692,Z 732.801,A -85,B 0,C 180,E1 27654.054,E2 27654.054} C_VEL
LIN {X 0,Y 577.292,Z 751.101,A -85,B 0,C 180,E1 27652.505,E2 27652.505} C_VEL
LIN {X 0,Y 576.929,Z 768.226,A -85,B 0,C 180,E1 27650.811,E2 27650.811} C_VEL
LIN {X 0,Y 576.628,Z 783.727,A -85,B 0,C 180,E1 27649.026,E2 27649.026} C_VEL
LIN {X 0,Y 576.388,Z 798.133,A -85,B 0,C 180,E1 27647.096,E2 27647.096} C_VEL
LIN {X 0,Y 576.223,Z 810.343,A -85,B 0,C 180,E1 27645.19,E2 27645.19} C_VEL
LIN {X 0,Y 576.083,Z 821.377,A -85,B 0,C 180,E1 27643.142,E2 27643.142} C_VEL
LIN {X 0,Y 575.997,Z 830.486,A -85,B 0,C 180,E1 27641.109,E2 27641.109} C_VEL
LIN {X 0,Y 575.956,Z 838.255,A -85,B 0,C 180,E1 27638.989,E2 27638.989} C_VEL
LIN {X 0,Y 575.931,Z 844.174,A -85,B 0,C 180,E1 27636.88,E2 27636.88} C_VEL
LIN {X 0,Y 575.916,Z 848.632,A -85,B 0,C 180,E1 27634.68,E2 27634.68} C_VEL
LIN {X 0,Y 575.908,Z 851.419,A -85,B 0,C 180,E1 27632.488,E2 27632.488} C_VEL
LIN {X 0,Y 575.9,Z 852.451,A -85,B 0,C 180,E1 27630.298,E2 27630.298} C_VEL
LIN {X 0,Y 575.907,Z 851.822,A -85,B 0,C 180,E1 27628.11,E2 27628.11} C_VEL
LIN {X 0,Y 575.913,Z 849.582,A -85,B 0,C 180,E1 27625.918,E2 27625.918} C_VEL
LIN {X 0,Y 575.917,Z 845.79,A -85,B 0,C 180,E1 27623.821,E2 27623.821} C_VEL
LIN {X 0,Y 575.939,Z 840.358,A -85,B 0,C 180,E1 27621.708,E2 27621.708} C_VEL
LIN {X 0,Y 575.982,Z 833.317,A -85,B 0,C 180,E1 27619.599,E2 27619.599} C_VEL
LIN {X 0,Y 576.047,Z 824.761,A -85,B 0,C 180,E1 27617.571,E2 27617.571} C_VEL
LIN {X 0,Y 576.162,Z 813.829,A -85,B 0,C 180,E1 27615.426,E2 27615.426} C_VEL
LIN {X 0,Y 576.34,Z 801.996,A -85,B 0,C 180,E1 27613.47,E2 27613.47} C_VEL
LIN {X 0,Y 576.568,Z 787.906,A -85,B 0,C 180,E1 27611.497,E2 27611.497} C_VEL
LIN {X 0,Y 576.845,Z 772.655,A -85,B 0,C 180,E1 27609.673,E2 27609.673} C_VEL
LIN {X 0,Y 577.16,Z 756.705,A -85,B 0,C 180,E1 27608.025,E2 27608.025} C_VEL
LIN {X 0,Y 577.539,Z 738.773,A -85,B 0,C 180,E1 27606.427,E2 27606.427} C_VEL
LIN {X 0,Y 577.963,Z 720.448,A -85,B 0,C 180,E1 27605.026,E2 27605.026} C_VEL
LIN {X 0,Y 578.38,Z 700.426,A -85,B 0,C 180,E1 27603.733,E2 27603.733} C_VEL
LIN {X 0,Y 578.753,Z 679.756,A -85,B 0,C 180,E1 27602.621,E2 27602.621} C_VEL
LIN {X 0,Y 579.17,Z 658.705,A -85,B 0,C 180,E1 27601.696,E2 27601.696} C_VEL
LIN {X 0,Y 579.503,Z 637.121,A -85,B 0,C 180,E1 27600.952,E2 27600.952} C_VEL
LIN {X 0,Y 579.737,Z 615.708,A -85,B 0,C 180,E1 27600.409,E2 27600.409} C_VEL
LIN {X 0,Y 579.933,Z 591.061,A -85,B 0,C 180,E1 27599.996,E2 27599.996} C_VEL
LIN {X 0,Y 580.757,Z 366.779,A -85,B 0,C 180,E1 27596.855,E2 27596.855} C_VEL
LIN {X 0,Y 580.854,Z 308.347,A -85,B 0,C 180,E1 27596.012,E2 27596.012} C_VEL
LIN {X 0,Y 579.698,Z 302.65,A -85,B 0,C 180,E1 27595.84,E2 27595.84} C_VEL
LIN {X 0,Y 580.326,Z 262.162,A -85,B 0,C 180,E1 27592.912,E2 27592.912} C_VEL
LIN {X 0,Y 580.333,Z 251.354,A -85,B 0,C 180,E1 27592.1,E2 27592.1} C_VEL
LIN {X 0,Y 577.033,Z 243.731,A -85,B 0,C 180,E1 27591.247,E2 27591.247} C_VEL
LIN {X 0,Y 579.23,Z 246.328,A -85,B 0,C 180,E1 27590.977,E2 27590.977} C_VEL
LIN {X 0,Y 580.886,Z 247.587,A -85,B 0,C 180,E1 27590.776,E2 27590.776} C_VEL
LIN {X 0,Y 583.588,Z 251.387,A -85,B 0,C 180,E1 27590.452,E2 27590.452} C_VEL
LIN {X 0,Y 585.977,Z 253.699,A -85,B 0,C 180,E1 27590.17,E2 27590.17} C_VEL
LIN {X 0,Y 586.862,Z 254.978,A -85,B 0,C 180,E1 27590.067,E2 27590.067} C_VEL
LIN {X 0,Y 587.045,Z 336.529,A -85,B 0,C 180,E1 27590.045,E2 27590.045} C_VEL
LIN {X 0,Y 588.185,Z 348.052,A -85,B 0,C 180,E1 27589.913,E2 27589.913} C_VEL
LIN {X 0,Y 590.323,Z 357.703,A -85,B 0,C 180,E1 27589.667,E2 27589.667} C_VEL
LIN {X 0,Y 593.406,Z 365.83,A -85,B 0,C 180,E1 27589.317,E2 27589.317} C_VEL
LIN {X 0,Y 595.523,Z 370.852,A -85,B 0,C 180,E1 27588.95,E2 27588.95} C_VEL
LIN {X 0,Y 596.641,Z 374.891,A -85,B 0,C 180,E1 27588.458,E2 27588.458} C_VEL
LIN {X 0,Y 596.603,Z 377.526,A -85,B 0,C 180,E1 27587.904,E2 27587.904} C_VEL
LIN {X 0,Y 595.531,Z 378.744,A -85,B 0,C 180,E1 27587.339,E2 27587.339} C_VEL
LIN {X 0,Y 593.761,Z 378.621,A -85,B 0,C 180,E1 27586.815,E2 27586.815} C_VEL
LIN {X 0,Y 591.079,Z 376.953,A -85,B 0,C 180,E1 27586.245,E2 27586.245} C_VEL
LIN {X 0,Y 587.973,Z 373.577,A -85,B 0,C 180,E1 27585.718,E2 27585.718} C_VEL
LIN {X 0,Y 584.374,Z 367.202,A -85,B 0,C 180,E1 27585.037,E2 27585.037} C_VEL
LIN {X 0,Y 581.757,Z 358.138,A -85,B 0,C 180,E1 27584.217,E2 27584.217} C_VEL
LIN {X 0,Y 580.423,Z 346.446,A -85,B 0,C 180,E1 27583.283,E2 27583.283} C_VEL
LIN {X 0,Y 581.062,Z 293.751,A -85,B 0,C 180,E1 27579.41,E2 27579.41} C_VEL
LIN {X 0,Y 581.829,Z 257.53,A -85,B 0,C 180,E1 27576.606,E2 27576.606} C_VEL
LIN {X 0,Y 581.877,Z 253.767,A -85,B 0,C 180,E1 27576.302,E2 27576.302} C_VEL
LIN {X 0,Y 577.452,Z 244.433,A -85,B 0,C 180,E1 27575.089,E2 27575.089} C_VEL
LIN {X 0,Y 576.132,Z 240.972,A -85,B 0,C 180,E1 27574.652,E2 27574.652} C_VEL
LIN {X 0,Y 576.145,Z 240.969,A -85,B 0,C 180,E1 27571.491,E2 27571.491} C_VEL
LIN {X 0,Y 576.143,Z 240.969,A -85,B 0,C 180,E1 27568.163,E2 27568.163} C_VEL
LIN {X 0,Y 576.187,Z 241.17,A -85,B 0,C 180,E1 27566.612,E2 27566.612} C_VEL
LIN {X 0,Y 576.571,Z 246.195,A -85,B 0,C 180,E1 27566.29,E2 27566.29} C_VEL
LIN {X 0,Y 577.049,Z 287.466,A -85,B 0,C 180,E1 27563.664,E2 27563.664} C_VEL
LIN {X 0,Y 577.428,Z 325.454,A -85,B 0,C 180,E1 27561.11,E2 27561.11} C_VEL
LIN {X 0,Y 577.407,Z 367.562,A -85,B 0,C 180,E1 27558.161,E2 27558.161} C_VEL
LIN {X 0,Y 577.033,Z 413.55,A -85,B 0,C 180,E1 27554.859,E2 27554.859} C_VEL
LIN {X 0,Y 576.682,Z 460.901,A -85,B 0,C 180,E1 27551.501,E2 27551.501} C_VEL
LIN {X 0,Y 576.561,Z 486.112,A -85,B 0,C 180,E1 27549.762,E2 27549.762} C_VEL
LIN {X 0,Y 576.6,Z 600.137,A -85,B 0,C 180,E1 27548.306,E2 27548.306} C_VEL
LIN {X 0,Y 576.507,Z 614.608,A -85,B 0,C 180,E1 27547.937,E2 27547.937} C_VEL
LIN {X 0,Y 576.412,Z 629.162,A -85,B 0,C 180,E1 27547.375,E2 27547.375} C_VEL
LIN {X 0,Y 576.292,Z 642.181,A -85,B 0,C 180,E1 27546.675,E2 27546.675} C_VEL
LIN {X 0,Y 576.203,Z 655.021,A -85,B 0,C 180,E1 27545.776,E2 27545.776} C_VEL
LIN {X 0,Y 576.102,Z 666.041,A -85,B 0,C 180,E1 27544.778,E2 27544.778} C_VEL
LIN {X 0,Y 576.031,Z 675.739,A -85,B 0,C 180,E1 27543.682,E2 27543.682} C_VEL
LIN {X 0,Y 575.975,Z 683.994,A -85,B 0,C 180,E1 27542.487,E2 27542.487} C_VEL
LIN {X 0,Y 575.941,Z 690.93,A -85,B 0,C 180,E1 27541.193,E2 27541.193} C_VEL
LIN {X 0,Y 575.925,Z 696.381,A -85,B 0,C 180,E1 27539.801,E2 27539.801} C_VEL
LIN {X 0,Y 575.918,Z 700.011,A -85,B 0,C 180,E1 27538.408,E2 27538.408} C_VEL
LIN {X 0,Y 575.916,Z 702.115,A -85,B 0,C 180,E1 27536.915,E2 27536.915} C_VEL
LIN {X 0,Y 575.918,Z 702.342,A -85,B 0,C 180,E1 27535.419,E2 27535.419} C_VEL
LIN {X 0,Y 575.917,Z 700.809,A -85,B 0,C 180,E1 27533.92,E2 27533.92} C_VEL
LIN {X 0,Y 575.922,Z 697.609,A -85,B 0,C 180,E1 27532.518,E2 27532.518} C_VEL
LIN {X 0,Y 575.935,Z 692.666,A -85,B 0,C 180,E1 27531.111,E2 27531.111} C_VEL
LIN {X 0,Y 575.965,Z 685.647,A -85,B 0,C 180,E1 27529.699,E2 27529.699} C_VEL
LIN {X 0,Y 576.016,Z 677.667,A -85,B 0,C 180,E1 27528.485,E2 27528.485} C_VEL
LIN {X 0,Y 576.097,Z 667.383,A -85,B 0,C 180,E1 27527.265,E2 27527.265} C_VEL
LIN {X 0,Y 576.178,Z 656.963,A -85,B 0,C 180,E1 27526.298,E2 27526.298} C_VEL
LIN {X 0,Y 576.27,Z 645.308,A -85,B 0,C 180,E1 27525.428,E2 27525.428} C_VEL
LIN {X 0,Y 576.288,Z 642.657,A -85,B 0,C 180,E1 27525.262,E2 27525.262} C_VEL
LIN {X 0,Y 575.518,Z 636.034,A -85,B 0,C 180,E1 27524.86,E2 27524.86} C_VEL
LIN {X 0,Y 571.195,Z 623.842,A -85,B 0,C 180,E1 27524.195,E2 27524.195} C_VEL
LIN {X 0,Y 569.118,Z 615.897,A -85,B 0,C 180,E1 27523.853,E2 27523.853} C_VEL
LIN {X 0,Y 568.685,Z 611.706,A -85,B 0,C 180,E1 27523.718,E2 27523.718} C_VEL
LIN {X 0,Y 568.793,Z 597.59,A -85,B 0,C 180,E1 27523.385,E2 27523.385} C_VEL
LIN {X 0,Y 568.763,Z 486.518,A -85,B 0,C 180,E1 27521.96,E2 27521.96} C_VEL
LIN {X 0,Y 568.674,Z 485.315,A -85,B 0,C 180,E1 27521.926,E2 27521.926} C_VEL
LIN {X 0,Y 569.064,Z 439.69,A -85,B 0,C 180,E1 27518.672,E2 27518.672} C_VEL
LIN {X 0,Y 569.522,Z 394.463,A -85,B 0,C 180,E1 27515.412,E2 27515.412} C_VEL
LIN {X 0,Y 569.948,Z 348.548,A -85,B 0,C 180,E1 27512.069,E2 27512.069} C_VEL
LIN {X 0,Y 570.07,Z 305.136,A -85,B 0,C 180,E1 27508.958,E2 27508.958} C_VEL
LIN {X 0,Y 570.043,Z 260.924,A -85,B 0,C 180,E1 27505.794,E2 27505.794} C_VEL
LIN {X 0,Y 569.916,Z 248.105,A -85,B 0,C 180,E1 27504.869,E2 27504.869} C_VEL
LIN {X 0,Y 568.217,Z 241.96,A -85,B 0,C 180,E1 27504.321,E2 27504.321} C_VEL
LIN {X 0,Y 568.191,Z 241.96,A -85,B 0,C 180,E1 27501.06,E2 27501.06} C_VEL
LIN {X 0,Y 568.221,Z 241.955,A -85,B 0,C 180,E1 27497.764,E2 27497.764} C_VEL
LIN {X 0,Y 568.22,Z 241.96,A -85,B 0,C 180,E1 27494.313,E2 27494.313} C_VEL
LIN {X 0,Y 568.184,Z 241.961,A -85,B 0,C 180,E1 27490.98,E2 27490.98} C_VEL
LIN {X 0,Y 568.208,Z 241.997,A -85,B 0,C 180,E1 27488.133,E2 27488.133} C_VEL
LIN {X 0,Y 570.199,Z 247.881,A -85,B 0,C 180,E1 27487.353,E2 27487.353} C_VEL
LIN {X 0,Y 571.885,Z 253.476,A -85,B 0,C 180,E1 27486.723,E2 27486.723} C_VEL
LIN {X 0,Y 571.192,Z 288.952,A -85,B 0,C 180,E1 27483.568,E2 27483.568} C_VEL
LIN {X 0,Y 571.114,Z 300.73,A -85,B 0,C 180,E1 27482.567,E2 27482.567} C_VEL
LIN {X 0,Y 572.629,Z 308.809,A -85,B 0,C 180,E1 27482.367,E2 27482.367} C_VEL
LIN {X 0,Y 571.724,Z 540.585,A -85,B 0,C 180,E1 27479.192,E2 27479.192} C_VEL
LIN {X 0,Y 571.533,Z 566.515,A -85,B 0,C 180,E1 27478.777,E2 27478.777} C_VEL
LIN {X 0,Y 571.255,Z 586.976,A -85,B 0,C 180,E1 27478.259,E2 27478.259} C_VEL
LIN {X 0,Y 570.963,Z 605.602,A -85,B 0,C 180,E1 27477.612,E2 27477.612} C_VEL
LIN {X 0,Y 570.594,Z 624.751,A -85,B 0,C 180,E1 27476.766,E2 27476.766} C_VEL
LIN {X 0,Y 570.176,Z 643.435,A -85,B 0,C 180,E1 27475.737,E2 27475.737} C_VEL
LIN {X 0,Y 569.769,Z 661.777,A -85,B 0,C 180,E1 27474.521,E2 27474.521} C_VEL
LIN {X 0,Y 569.363,Z 678.829,A -85,B 0,C 180,E1 27473.164,E2 27473.164} C_VEL
LIN {X 0,Y 569.013,Z 694.472,A -85,B 0,C 180,E1 27471.709,E2 27471.709} C_VEL
LIN {X 0,Y 568.678,Z 709.508,A -85,B 0,C 180,E1 27470.051,E2 27470.051} C_VEL
LIN {X 0,Y 568.43,Z 722.642,A -85,B 0,C 180,E1 27468.352,E2 27468.352} C_VEL
LIN {X 0,Y 568.228,Z 734.993,A -85,B 0,C 180,E1 27466.457,E2 27466.457} C_VEL
LIN {X 0,Y 568.08,Z 744.601,A -85,B 0,C 180,E1 27464.682,E2 27464.682} C_VEL
LIN {X 0,Y 567.994,Z 753.471,A -85,B 0,C 180,E1 27462.712,E2 27462.712} C_VEL
LIN {X 0,Y 567.948,Z 760.457,A -85,B 0,C 180,E1 27460.755,E2 27460.755} C_VEL
LIN {X 0,Y 567.925,Z 765.757,A -85,B 0,C 180,E1 27458.811,E2 27458.811} C_VEL
LIN {X 0,Y 567.916,Z 769.783,A -85,B 0,C 180,E1 27456.673,E2 27456.673} C_VEL
LIN {X 0,Y 567.909,Z 771.893,A -85,B 0,C 180,E1 27454.645,E2 27454.645} C_VEL
LIN {X 0,Y 567.901,Z 772.423,A -85,B 0,C 180,E1 27452.523,E2 27452.523} C_VEL
LIN {X 0,Y 567.901,Z 771.301,A -85,B 0,C 180,E1 27450.504,E2 27450.504} C_VEL
LIN {X 0,Y 567.905,Z 768.588,A -85,B 0,C 180,E1 27448.487,E2 27448.487} C_VEL
LIN {X 0,Y 567.926,Z 763.954,A -85,B 0,C 180,E1 27446.366,E2 27446.366} C_VEL
LIN {X 0,Y 567.965,Z 757.752,A -85,B 0,C 180,E1 27444.342,E2 27444.342} C_VEL
LIN {X 0,Y 568.033,Z 749.26,A -85,B 0,C 180,E1 27442.21,E2 27442.21} C_VEL
LIN {X 0,Y 568.147,Z 739.657,A -85,B 0,C 180,E1 27440.273,E2 27440.273} C_VEL
LIN {X 0,Y 568.331,Z 727.895,A -85,B 0,C 180,E1 27438.327,E2 27438.327} C_VEL
LIN {X 0,Y 568.55,Z 716.124,A -85,B 0,C 180,E1 27436.681,E2 27436.681} C_VEL
LIN {X 0,Y 568.86,Z 701.333,A -85,B 0,C 180,E1 27434.922,E2 27434.922} C_VEL
LIN {X 0,Y 569.191,Z 686.309,A -85,B 0,C 180,E1 27433.414,E2 27433.414} C_VEL
LIN {X 0,Y 569.608,Z 669.002,A -85,B 0,C 180,E1 27431.932,E2 27431.932} C_VEL
LIN {X 0,Y 569.996,Z 651.612,A -85,B 0,C 180,E1 27430.69,E2 27430.69} C_VEL
LIN {X 0,Y 570.401,Z 633.232,A -85,B 0,C 180,E1 27429.584,E2 27429.584} C_VEL
LIN {X 0,Y 570.798,Z 613.658,A -85,B 0,C 180,E1 27428.632,E2 27428.632} C_VEL
LIN {X 0,Y 571.167,Z 594.559,A -85,B 0,C 180,E1 27427.891,E2 27427.891} C_VEL
LIN {X 0,Y 571.448,Z 573.602,A -85,B 0,C 180,E1 27427.289,E2 27427.289} C_VEL
LIN {X 0,Y 571.643,Z 553.976,A -85,B 0,C 180,E1 27426.907,E2 27426.907} C_VEL
LIN {X 0,Y 572.646,Z 312.346,A -85,B 0,C 180,E1 27423.594,E2 27423.594} C_VEL
LIN {X 0,Y 572.426,Z 304.831,A -85,B 0,C 180,E1 27423.475,E2 27423.475} C_VEL
LIN {X 0,Y 571.363,Z 299.187,A -85,B 0,C 180,E1 27423.329,E2 27423.329} C_VEL
LIN {X 0,Y 572.128,Z 255.098,A -85,B 0,C 180,E1 27420.012,E2 27420.012} C_VEL
LIN {X 0,Y 572.109,Z 252.867,A -85,B 0,C 180,E1 27419.837,E2 27419.837} C_VEL
LIN {X 0,Y 568.223,Z 241.959,A -85,B 0,C 180,E1 27418.699,E2 27418.699} C_VEL
LIN {X 0,Y 568.216,Z 241.961,A -85,B 0,C 180,E1 27415.241,E2 27415.241} C_VEL
LIN {X 0,Y 568.219,Z 241.962,A -85,B 0,C 180,E1 27411.728,E2 27411.728} C_VEL
LIN {X 0,Y 568.223,Z 241.959,A -85,B 0,C 180,E1 27408.307,E2 27408.307} C_VEL
LIN {X 0,Y 568.199,Z 241.959,A -85,B 0,C 180,E1 27404.976,E2 27404.976} C_VEL
LIN {X 0,Y 568.198,Z 241.958,A -85,B 0,C 180,E1 27401.745,E2 27401.745} C_VEL
LIN {X 0,Y 568.22,Z 241.957,A -85,B 0,C 180,E1 27398.46,E2 27398.46} C_VEL
LIN {X 0,Y 568.218,Z 241.959,A -85,B 0,C 180,E1 27395.005,E2 27395.005} C_VEL
LIN {X 0,Y 568.218,Z 241.96,A -85,B 0,C 180,E1 27391.508,E2 27391.508} C_VEL
LIN {X 0,Y 568.203,Z 241.96,A -85,B 0,C 180,E1 27388.253,E2 27388.253} C_VEL
LIN {X 0,Y 568.221,Z 242.122,A -85,B 0,C 180,E1 27387.127,E2 27387.127} C_VEL
LIN {X 0,Y 570.231,Z 249.649,A -85,B 0,C 180,E1 27386.447,E2 27386.447} C_VEL
LIN {X 0,Y 570.221,Z 294.17,A -85,B 0,C 180,E1 27382.99,E2 27382.99} C_VEL
LIN {X 0,Y 570.065,Z 334.657,A -85,B 0,C 180,E1 27379.84,E2 27379.84} C_VEL
LIN {X 0,Y 569.649,Z 375.839,A -85,B 0,C 180,E1 27376.593,E2 27376.593} C_VEL
LIN {X 0,Y 569.155,Z 419.227,A -85,B 0,C 180,E1 27373.202,E2 27373.202} C_VEL
LIN {X 0,Y 569.026,Z 436.455,A -85,B 0,C 180,E1 27371.897,E2 27371.897} C_VEL
LIN {X 0,Y 569.481,Z 444.022,A -85,B 0,C 180,E1 27371.786,E2 27371.786} C_VEL
LIN {X 0,Y 569.153,Z 578.267,A -85,B 0,C 180,E1 27370.042,E2 27370.042} C_VEL
LIN {X 0,Y 569.045,Z 594.978,A -85,B 0,C 180,E1 27369.635,E2 27369.635} C_VEL
LIN {X 0,Y 568.891,Z 609.426,A -85,B 0,C 180,E1 27369.102,E2 27369.102} C_VEL
LIN {X 0,Y 568.737,Z 623.038,A -85,B 0,C 180,E1 27368.442,E2 27368.442} C_VEL
LIN {X 0,Y 568.535,Z 637.566,A -85,B 0,C 180,E1 27367.529,E2 27367.529} C_VEL
LIN {X 0,Y 568.377,Z 649.695,A -85,B 0,C 180,E1 27366.566,E2 27366.566} C_VEL
LIN {X 0,Y 568.237,Z 661.224,A -85,B 0,C 180,E1 27365.453,E2 27365.453} C_VEL
